LIN {X 0,Y 314.048,Z 563.182,A -85,B 0,C 180,E1 -16082.332,E2 -16082.332} C_VEL
LIN {X 0,Y 311.927,Z 573.073,A -85,B 0,C 180,E1 -16084.18,E2 -16084.18} C_VEL
LIN {X 0,Y 309.879,Z 582.152,A -85,B 0,C 180,E1 -16086.262,E2 -16086.262} C_VEL
LIN {X 0,Y 307.951,Z 590.287,A -85,B 0,C 180,E1 -16088.584,E2 -16088.584} C_VEL
LIN {X 0,Y 306.633,Z 595.997,A -85,B 0,C 180,E1 -16090.59,E2 -16090.59} C_VEL
LIN {X 0,Y 305.291,Z 601.948,A -85,B 0,C 180,E1 -16093.277,E2 -16093.277} C_VEL
LIN {X 0,Y 304.462,Z 606.083,A -85,B 0,C 180,E1 -16095.816,E2 -16095.816} C_VEL
LIN {X 0,Y 303.923,Z 608.604,A -85,B 0,C 180,E1 -16097.988,E2 -16097.988} C_VEL
LIN {X 0,Y 303.601,Z 610.421,A -85,B 0,C 180,E1 -16100.675,E2 -16100.675} C_VEL
LIN {X 0,Y 303.604,Z 610.898,A -85,B 0,C 180,E1 -16103.354,E2 -16103.354} C_VEL
LIN {X 0,Y 303.641,Z 610.642,A -85,B 0,C 180,E1 -16104.688,E2 -16104.688} C_VEL
LIN {X 0,Y 303.656,Z 609.146,A -85,B 0,C 180,E1 -16107.347,E2 -16107.347} C_VEL
LIN {X 0,Y 303.822,Z 606.306,A -85,B 0,C 180,E1 -16110,E2 -16110} C_VEL
LIN {X 0,Y 304.271,Z 602.046,A -85,B 0,C 180,E1 -16112.648,E2 -16112.648} C_VEL
LIN {X 0,Y 305.064,Z 596.235,A -85,B 0,C 180,E1 -16115.287,E2 -16115.287} C_VEL
LIN {X 0,Y 306.201,Z 589.686,A -85,B 0,C 180,E1 -16117.584,E2 -16117.584} C_VEL
LIN {X 0,Y 307.622,Z 581.561,A -85,B 0,C 180,E1 -16119.866,E2 -16119.866} C_VEL
LIN {X 0,Y 309.146,Z 572.018,A -85,B 0,C 180,E1 -16122.027,E2 -16122.027} C_VEL
LIN {X 0,Y 310.712,Z 562.821,A -85,B 0,C 180,E1 -16123.739,E2 -16123.739} C_VEL
LIN {X 0,Y 312.561,Z 551.345,A -85,B 0,C 180,E1 -16125.486,E2 -16125.486} C_VEL
LIN {X 0,Y 314.206,Z 539.898,A -85,B 0,C 180,E1 -16126.904,E2 -16126.904} C_VEL
LIN {X 0,Y 315.826,Z 527.334,A -85,B 0,C 180,E1 -16128.151,E2 -16128.151} C_VEL
LIN {X 0,Y 317.303,Z 514.341,A -85,B 0,C 180,E1 -16129.152,E2 -16129.152} C_VEL
LIN {X 0,Y 318.433,Z 500.352,A -85,B 0,C 180,E1 -16129.962,E2 -16129.962} C_VEL
LIN {X 0,Y 319.213,Z 486.734,A -85,B 0,C 180,E1 -16130.499,E2 -16130.499} C_VEL
LIN {X 0,Y 321.884,Z 387.028,A -85,B 0,C 180,E1 -16132.739,E2 -16132.739} C_VEL
LIN {X 0,Y 315.759,Z 371.085,A -85,B 0,C 180,E1 -16133.694,E2 -16133.694} C_VEL
LIN {X 0,Y 308.735,Z 355.109,A -85,B 0,C 180,E1 -16134.786,E2 -16134.786} C_VEL
LIN {X 0,Y 306.421,Z 349.762,A -85,B 0,C 180,E1 -16135.185,E2 -16135.185} C_VEL
LIN {X 0,Y 305.544,Z 346.052,A -85,B 0,C 180,E1 -16136.413,E2 -16136.413} C_VEL
LIN {X 0,Y 305.46,Z 346.061,A -85,B 0,C 180,E1 -16140.408,E2 -16140.408} C_VEL
LIN {X 0,Y 305.438,Z 346.062,A -85,B 0,C 180,E1 -16141.171,E2 -16141.171} C_VEL
LIN {X 0,Y 304.797,Z 346.144,A -85,B 0,C 180,E1 -16142.272,E2 -16142.272} C_VEL
LIN {X 0,Y 302.003,Z 346.49,A -85,B 0,C 180,E1 -16144.064,E2 -16144.064} C_VEL
LIN {X 0,Y 299.606,Z 346.785,A -85,B 0,C 180,E1 -16145.518,E2 -16145.518} C_VEL
LIN {X 0,Y 298.55,Z 346.917,A -85,B 0,C 180,E1 -16146.642,E2 -16146.642} C_VEL
LIN {X 0,Y 298.45,Z 346.93,A -85,B 0,C 180,E1 -16147.024,E2 -16147.024} C_VEL
LIN {X 0,Y 298.383,Z 346.926,A -85,B 0,C 180,E1 -16151.26,E2 -16151.26} C_VEL
LIN {X 0,Y 298.352,Z 346.941,A -85,B 0,C 180,E1 -16155.034,E2 -16155.034} C_VEL
LIN {X 0,Y 298.381,Z 346.935,A -85,B 0,C 180,E1 -16158.737,E2 -16158.737} C_VEL
LIN {X 0,Y 298.404,Z 346.93,A -85,B 0,C 180,E1 -16162.24,E2 -16162.24} C_VEL
LIN {X 0,Y 298.404,Z 346.935,A -85,B 0,C 180,E1 -16165.58,E2 -16165.58} C_VEL
LIN {X 0,Y 298.386,Z 346.941,A -85,B 0,C 180,E1 -16168.789,E2 -16168.789} C_VEL
LIN {X 0,Y 298.438,Z 346.919,A -85,B 0,C 180,E1 -16171.901,E2 -16171.901} C_VEL
LIN {X 0,Y 298.459,Z 346.929,A -85,B 0,C 180,E1 -16174.921,E2 -16174.921} C_VEL
LIN {X 0,Y 298.41,Z 346.918,A -85,B 0,C 180,E1 -16179.312,E2 -16179.312} C_VEL
LIN {X 0,Y 298.458,Z 346.927,A -85,B 0,C 180,E1 -16182.174,E2 -16182.174} C_VEL
LIN {X 0,Y 298.579,Z 346.911,A -85,B 0,C 180,E1 -16184.993,E2 -16184.993} C_VEL
LIN {X 0,Y 298.574,Z 346.907,A -85,B 0,C 180,E1 -16189.145,E2 -16189.145} C_VEL
LIN {X 0,Y 298.707,Z 346.9,A -85,B 0,C 180,E1 -16191.884,E2 -16191.884} C_VEL
LIN {X 0,Y 298.628,Z 346.89,A -85,B 0,C 180,E1 -16194.598,E2 -16194.598} C_VEL
LIN {X 0,Y 298.893,Z 346.877,A -85,B 0,C 180,E1 -16198.652,E2 -16198.652} C_VEL
LIN {X 0,Y 298.898,Z 346.872,A -85,B 0,C 180,E1 -16201.347,E2 -16201.347} C_VEL
LIN {X 0,Y 298.722,Z 346.899,A -85,B 0,C 180,E1 -16206.755,E2 -16206.755} C_VEL
LIN {X 0,Y 298.616,Z 346.897,A -85,B 0,C 180,E1 -16209.482,E2 -16209.482} C_VEL
LIN {X 0,Y 298.534,Z 346.922,A -85,B 0,C 180,E1 -16213.616,E2 -16213.616} C_VEL
LIN {X 0,Y 298.477,Z 346.92,A -85,B 0,C 180,E1 -16216.412,E2 -16216.412} C_VEL
LIN {X 0,Y 298.474,Z 346.929,A -85,B 0,C 180,E1 -16219.639,E2 -16219.639} C_VEL
LIN {X 0,Y 298.415,Z 346.935,A -85,B 0,C 180,E1 -16223.601,E2 -16223.601} C_VEL
LIN {X 0,Y 298.4,Z 346.931,A -85,B 0,C 180,E1 -16226.583,E2 -16226.583} C_VEL
LIN {X 0,Y 298.385,Z 346.937,A -85,B 0,C 180,E1 -16229.644,E2 -16229.644} C_VEL
LIN {X 0,Y 298.385,Z 346.94,A -85,B 0,C 180,E1 -16232.801,E2 -16232.801} C_VEL
LIN {X 0,Y 298.44,Z 346.932,A -85,B 0,C 180,E1 -16236.808,E2 -16236.808} C_VEL
LIN {X 0,Y 298.38,Z 346.928,A -85,B 0,C 180,E1 -16241.088,E2 -16241.088} C_VEL
LIN {X 0,Y 298.393,Z 346.937,A -85,B 0,C 180,E1 -16243.104,E2 -16243.104} C_VEL
LIN {X 0,Y 298.398,Z 346.939,A -85,B 0,C 180,E1 -16246.921,E2 -16246.921} C_VEL
LIN {X 0,Y 298.399,Z 346.946,A -85,B 0,C 180,E1 -16251.007,E2 -16251.007} C_VEL
LIN {X 0,Y 298.446,Z 347.048,A -85,B 0,C 180,E1 -16253.151,E2 -16253.151} C_VEL
LIN {X 0,Y 301.507,Z 359.563,A -85,B 0,C 180,E1 -16257.05,E2 -16257.05} C_VEL
LIN {X 0,Y 302.652,Z 364.595,A -85,B 0,C 180,E1 -16258.477,E2 -16258.477} C_VEL
LIN {X 0,Y 310.44,Z 383.686,A -85,B 0,C 180,E1 -16259.756,E2 -16259.756} C_VEL
LIN {X 0,Y 314.914,Z 411.594,A -85,B 0,C 180,E1 -16260.88,E2 -16260.88} C_VEL
LIN {X 0,Y 312.457,Z 500.646,A -85,B 0,C 180,E1 -16262.905,E2 -16262.905} C_VEL
LIN {X 0,Y 311.58,Z 514.525,A -85,B 0,C 180,E1 -16263.411,E2 -16263.411} C_VEL
LIN {X 0,Y 310.308,Z 528.189,A -85,B 0,C 180,E1 -16264.153,E2 -16264.153} C_VEL
LIN {X 0,Y 308.888,Z 541.031,A -85,B 0,C 180,E1 -16265.108,E2 -16265.108} C_VEL
LIN {X 0,Y 307.067,Z 554.478,A -85,B 0,C 180,E1 -16266.409,E2 -16266.409} C_VEL
LIN {X 0,Y 305.262,Z 566.32,A -85,B 0,C 180,E1 -16267.853,E2 -16267.853} C_VEL
LIN {X 0,Y 303.49,Z 576.274,A -85,B 0,C 180,E1 -16269.321,E2 -16269.321} C_VEL
LIN {X 0,Y 301.572,Z 587.25,A -85,B 0,C 180,E1 -16271.311,E2 -16271.311} C_VEL
LIN {X 0,Y 300.075,Z 596.312,A -85,B 0,C 180,E1 -16273.328,E2 -16273.328} C_VEL
LIN {X 0,Y 298.965,Z 603.853,A -85,B 0,C 180,E1 -16275.363,E2 -16275.363} C_VEL
LIN {X 0,Y 297.819,Z 611.042,A -85,B 0,C 180,E1 -16277.738,E2 -16277.738} C_VEL
LIN {X 0,Y 297.13,Z 616.051,A -85,B 0,C 180,E1 -16279.782,E2 -16279.782} C_VEL
LIN {X 0,Y 296.737,Z 621.214,A -85,B 0,C 180,E1 -16282.515,E2 -16282.515} C_VEL
LIN {X 0,Y 296.554,Z 624.106,A -85,B 0,C 180,E1 -16284.561,E2 -16284.561} C_VEL
LIN {X 0,Y 296.536,Z 626.656,A -85,B 0,C 180,E1 -16287.283,E2 -16287.283} C_VEL
LIN {X 0,Y 296.518,Z 627.833,A -85,B 0,C 180,E1 -16290,E2 -16290} C_VEL
LIN {X 0,Y 296.522,Z 627.671,A -85,B 0,C 180,E1 -16292.717,E2 -16292.717} C_VEL
LIN {X 0,Y 296.545,Z 626.116,A -85,B 0,C 180,E1 -16295.509,E2 -16295.509} C_VEL
LIN {X 0,Y 296.85,Z 623.32,A -85,B 0,C 180,E1 -16298.166,E2 -16298.166} C_VEL
LIN {X 0,Y 297.49,Z 619.034,A -85,B 0,C 180,E1 -16300.894,E2 -16300.894} C_VEL
LIN {X 0,Y 298.327,Z 614.817,A -85,B 0,C 180,E1 -16302.932,E2 -16302.932} C_VEL
LIN {X 0,Y 299.44,Z 609.647,A -85,B 0,C 180,E1 -16304.961,E2 -16304.961} C_VEL
LIN {X 0,Y 301.064,Z 602.238,A -85,B 0,C 180,E1 -16307.315,E2 -16307.315} C_VEL
LIN {X 0,Y 303.272,Z 593.049,A -85,B 0,C 180,E1 -16309.634,E2 -16309.634} C_VEL
LIN {X 0,Y 305.521,Z 583.471,A -85,B 0,C 180,E1 -16311.595,E2 -16311.595} C_VEL
LIN {X 0,Y 307.96,Z 572.871,A -85,B 0,C 180,E1 -16313.36,E2 -16313.36} C_VEL
LIN {X 0,Y 310.301,Z 561.536,A -85,B 0,C 180,E1 -16314.899,E2 -16314.899} C_VEL
LIN {X 0,Y 312.451,Z 549.755,A -85,B 0,C 180,E1 -16316.194,E2 -16316.194} C_VEL
LIN {X 0,Y 314.351,Z 537.392,A -85,B 0,C 180,E1 -16317.278,E2 -16317.278} C_VEL
LIN {X 0,Y 316.259,Z 523.679,A -85,B 0,C 180,E1 -16318.178,E2 -16318.178} C_VEL
LIN {X 0,Y 317.738,Z 509.393,A -85,B 0,C 180,E1 -16318.846,E2 -16318.846} C_VEL
LIN {X 0,Y 318.543,Z 494.481,A -85,B 0,C 180,E1 -16319.294,E2 -16319.294} C_VEL
LIN {X 0,Y 321.296,Z 414.11,A -85,B 0,C 180,E1 -16321.078,E2 -16321.078} C_VEL
LIN {X 0,Y 317.583,Z 394.103,A -85,B 0,C 180,E1 -16322.056,E2 -16322.056} C_VEL
LIN {X 0,Y 310.883,Z 379.558,A -85,B 0,C 180,E1 -16323.308,E2 -16323.308} C_VEL
LIN {X 0,Y 304.459,Z 366.874,A -85,B 0,C 180,E1 -16324.545,E2 -16324.545} C_VEL
LIN {X 0,Y 303.009,Z 363.713,A -85,B 0,C 180,E1 -16324.868,E2 -16324.868} C_VEL
LIN {X 0,Y 300.803,Z 355.353,A -85,B 0,C 180,E1 -16327.732,E2 -16327.732} C_VEL
LIN {X 0,Y 298.389,Z 346.922,A -85,B 0,C 180,E1 -16330.868,E2 -16330.868} C_VEL
LIN {X 0,Y 298.394,Z 346.931,A -85,B 0,C 180,E1 -16333.103,E2 -16333.103} C_VEL
LIN {X 0,Y 298.398,Z 346.935,A -85,B 0,C 180,E1 -16336.92,E2 -16336.92} C_VEL
LIN {X 0,Y 298.398,Z 346.941,A -85,B 0,C 180,E1 -16341.006,E2 -16341.006} C_VEL
LIN {X 0,Y 298.412,Z 346.941,A -85,B 0,C 180,E1 -16343.93,E2 -16343.93} C_VEL
LIN {X 0,Y 298.381,Z 346.932,A -85,B 0,C 180,E1 -16347.985,E2 -16347.985} C_VEL
LIN {X 0,Y 298.401,Z 346.924,A -85,B 0,C 180,E1 -16351.898,E2 -16351.898} C_VEL
LIN {X 0,Y 298.431,Z 346.929,A -85,B 0,C 180,E1 -16354.92,E2 -16354.92} C_VEL
LIN {X 0,Y 298.399,Z 346.94,A -85,B 0,C 180,E1 -16357.862,E2 -16357.862} C_VEL
LIN {X 0,Y 298.495,Z 346.926,A -85,B 0,C 180,E1 -16360.754,E2 -16360.754} C_VEL
LIN {X 0,Y 298.578,Z 346.913,A -85,B 0,C 180,E1 -16364.994,E2 -16364.994} C_VEL
LIN {X 0,Y 298.571,Z 346.91,A -85,B 0,C 180,E1 -16369.146,E2 -16369.146} C_VEL
LIN {X 0,Y 298.688,Z 346.898,A -85,B 0,C 180,E1 -16371.884,E2 -16371.884} C_VEL
LIN {X 0,Y 298.618,Z 346.91,A -85,B 0,C 180,E1 -16374.599,E2 -16374.599} C_VEL
LIN {X 0,Y 298.904,Z 346.869,A -85,B 0,C 180,E1 -16378.653,E2 -16378.653} C_VEL
LIN {X 0,Y 298.894,Z 346.874,A -85,B 0,C 180,E1 -16381.348,E2 -16381.348} C_VEL
LIN {X 0,Y 298.738,Z 346.89,A -85,B 0,C 180,E1 -16386.756,E2 -16386.756} C_VEL
LIN {X 0,Y 298.617,Z 346.915,A -85,B 0,C 180,E1 -16389.483,E2 -16389.483} C_VEL
LIN {X 0,Y 298.537,Z 346.923,A -85,B 0,C 180,E1 -16393.617,E2 -16393.617} C_VEL
LIN {X 0,Y 298.476,Z 346.921,A -85,B 0,C 180,E1 -16396.413,E2 -16396.413} C_VEL
LIN {X 0,Y 298.439,Z 346.931,A -85,B 0,C 180,E1 -16399.62,E2 -16399.62} C_VEL
LIN {X 0,Y 298.423,Z 346.933,A -85,B 0,C 180,E1 -16403.601,E2 -16403.601} C_VEL
LIN {X 0,Y 298.481,Z 346.932,A -85,B 0,C 180,E1 -16406.576,E2 -16406.576} C_VEL
LIN {X 0,Y 298.412,Z 346.938,A -85,B 0,C 180,E1 -16409.643,E2 -16409.643} C_VEL
LIN {X 0,Y 298.39,Z 346.942,A -85,B 0,C 180,E1 -16412.802,E2 -16412.802} C_VEL
LIN {X 0,Y 298.442,Z 346.929,A -85,B 0,C 180,E1 -16416.809,E2 -16416.809} C_VEL
LIN {X 0,Y 298.385,Z 346.943,A -85,B 0,C 180,E1 -16421.089,E2 -16421.089} C_VEL
LIN {X 0,Y 298.397,Z 346.939,A -85,B 0,C 180,E1 -16423.105,E2 -16423.105} C_VEL
LIN {X 0,Y 298.442,Z 347.061,A -85,B 0,C 180,E1 -16427.292,E2 -16427.292} C_VEL
LIN {X 0,Y 299.426,Z 350.748,A -85,B 0,C 180,E1 -16428.686,E2 -16428.686} C_VEL
LIN {X 0,Y 309.463,Z 368.66,A -85,B 0,C 180,E1 -16430.634,E2 -16430.634} C_VEL
LIN {X 0,Y 315.822,Z 381.45,A -85,B 0,C 180,E1 -16431.82,E2 -16431.82} C_VEL
LIN {X 0,Y 321.871,Z 395.005,A -85,B 0,C 180,E1 -16432.925,E2 -16432.925} C_VEL
LIN {X 0,Y 318.622,Z 487.207,A -85,B 0,C 180,E1 -16435.007,E2 -16435.007} C_VEL
LIN {X 0,Y 317.575,Z 501.841,A -85,B 0,C 180,E1 -16435.598,E2 -16435.598} C_VEL
LIN {X 0,Y 316.089,Z 515.831,A -85,B 0,C 180,E1 -16436.423,E2 -16436.423} C_VEL
LIN {X 0,Y 314.408,Z 527.939,A -85,B 0,C 180,E1 -16437.367,E2 -16437.367} C_VEL
LIN {X 0,Y 312.253,Z 540.703,A -85,B 0,C 180,E1 -16438.636,E2 -16438.636} C_VEL
LIN {X 0,Y 309.916,Z 552.287,A -85,B 0,C 180,E1 -16440.074,E2 -16440.074} C_VEL
LIN {X 0,Y 307.656,Z 562.893,A -85,B 0,C 180,E1 -16441.706,E2 -16441.706} C_VEL
LIN {X 0,Y 305.594,Z 572.086,A -85,B 0,C 180,E1 -16443.43,E2 -16443.43} C_VEL
LIN {X 0,Y 303.647,Z 580.667,A -85,B 0,C 180,E1 -16445.38,E2 -16445.38} C_VEL
LIN {X 0,Y 301.738,Z 588.045,A -85,B 0,C 180,E1 -16447.4,E2 -16447.4} C_VEL
LIN {X 0,Y 300.276,Z 594.164,A -85,B 0,C 180,E1 -16449.447,E2 -16449.447} C_VEL
LIN {X 0,Y 298.67,Z 600.637,A -85,B 0,C 180,E1 -16452.188,E2 -16452.188} C_VEL
LIN {X 0,Y 297.606,Z 605.444,A -85,B 0,C 180,E1 -16454.944,E2 -16454.944} C_VEL
LIN {X 0,Y 296.909,Z 608.73,A -85,B 0,C 180,E1 -16457.7,E2 -16457.7} C_VEL
LIN {X 0,Y 296.52,Z 610.594,A -85,B 0,C 180,E1 -16460.45,E2 -16460.45} C_VEL
LIN {X 0,Y 296.517,Z 611.111,A -85,B 0,C 180,E1 -16463.194,E2 -16463.194} C_VEL
LIN {X 0,Y 296.555,Z 610.874,A -85,B 0,C 180,E1 -16464.561,E2 -16464.561} C_VEL
LIN {X 0,Y 296.579,Z 609.417,A -85,B 0,C 180,E1 -16467.284,E2 -16467.284} C_VEL
LIN {X 0,Y 296.726,Z 606.619,A -85,B 0,C 180,E1 -16470,E2 -16470} C_VEL
LIN {X 0,Y 297.148,Z 603.624,A -85,B 0,C 180,E1 -16472.033,E2 -16472.033} C_VEL
LIN {X 0,Y 297.896,Z 598.23,A -85,B 0,C 180,E1 -16474.736,E2 -16474.736} C_VEL
LIN {X 0,Y 298.575,Z 593.122,A -85,B 0,C 180,E1 -16476.759,E2 -16476.759} C_VEL
LIN {X 0,Y 300.025,Z 585.752,A -85,B 0,C 180,E1 -16479.097,E2 -16479.097} C_VEL
LIN {X 0,Y 301.612,Z 576.798,A -85,B 0,C 180,E1 -16481.382,E2 -16481.382} C_VEL
LIN {X 0,Y 303.21,Z 567.089,A -85,B 0,C 180,E1 -16483.402,E2 -16483.402} C_VEL
LIN {X 0,Y 305.03,Z 556.516,A -85,B 0,C 180,E1 -16485.193,E2 -16485.193} C_VEL
LIN {X 0,Y 306.934,Z 544.818,A -85,B 0,C 180,E1 -16486.802,E2 -16486.802} C_VEL
LIN {X 0,Y 308.525,Z 533.376,A -85,B 0,C 180,E1 -16488.081,E2 -16488.081} C_VEL
LIN {X 0,Y 310.089,Z 520.948,A -85,B 0,C 180,E1 -16489.185,E2 -16489.185} C_VEL
LIN {X 0,Y 311.431,Z 507.132,A -85,B 0,C 180,E1 -16490.129,E2 -16490.129} C_VEL
LIN {X 0,Y 312.498,Z 493.489,A -85,B 0,C 180,E1 -16490.788,E2 -16490.788} C_VEL
LIN {X 0,Y 313.003,Z 479.899,A -85,B 0,C 180,E1 -16491.222,E2 -16491.222} C_VEL
LIN {X 0,Y 315.427,Z 388.282,A -85,B 0,C 180,E1 -16493.293,E2 -16493.293} C_VEL
LIN {X 0,Y 307.234,Z 367.72,A -85,B 0,C 180,E1 -16494.609,E2 -16494.609} C_VEL
LIN {X 0,Y 299.236,Z 349.982,A -85,B 0,C 180,E1 -16495.937,E2 -16495.937} C_VEL
LIN {X 0,Y 298.479,Z 346.931,A -85,B 0,C 180,E1 -16497.018,E2 -16497.018} C_VEL
LIN {X 0,Y 298.393,Z 346.94,A -85,B 0,C 180,E1 -16501.208,E2 -16501.208} C_VEL
LIN {X 0,Y 298.428,Z 346.933,A -85,B 0,C 180,E1 -16504.486,E2 -16504.486} C_VEL
LIN {X 0,Y 298.45,Z 346.93,A -85,B 0,C 180,E1 -16507.024,E2 -16507.024} C_VEL
LIN {X 0,Y 297.738,Z 347.023,A -85,B 0,C 180,E1 -16508.15,E2 -16508.15} C_VEL
LIN {X 0,Y 294.851,Z 347.382,A -85,B 0,C 180,E1 -16509.983,E2 -16509.983} C_VEL
LIN {X 0,Y 292.426,Z 347.682,A -85,B 0,C 180,E1 -16511.47,E2 -16511.47} C_VEL
LIN {X 0,Y 291.385,Z 347.812,A -85,B 0,C 180,E1 -16512.623,E2 -16512.623} C_VEL
LIN {X 0,Y 291.299,Z 347.821,A -85,B 0,C 180,E1 -16513.013,E2 -16513.013} C_VEL
LIN {X 0,Y 291.317,Z 347.818,A -85,B 0,C 180,E1 -16517.506,E2 -16517.506} C_VEL
LIN {X 0,Y 291.344,Z 347.817,A -85,B 0,C 180,E1 -16521.156,E2 -16521.156} C_VEL
LIN {X 0,Y 291.357,Z 347.817,A -85,B 0,C 180,E1 -16524.625,E2 -16524.625} C_VEL
LIN {X 0,Y 291.366,Z 347.814,A -85,B 0,C 180,E1 -16527.949,E2 -16527.949} C_VEL
LIN {X 0,Y 291.365,Z 347.805,A -85,B 0,C 180,E1 -16531.156,E2 -16531.156} C_VEL
LIN {X 0,Y 291.394,Z 347.805,A -85,B 0,C 180,E1 -16534.269,E2 -16534.269} C_VEL
LIN {X 0,Y 291.361,Z 347.811,A -85,B 0,C 180,E1 -16537.297,E2 -16537.297} C_VEL
LIN {X 0,Y 291.384,Z 347.793,A -85,B 0,C 180,E1 -16540.264,E2 -16540.264} C_VEL
LIN {X 0,Y 291.491,Z 347.797,A -85,B 0,C 180,E1 -16544.664,E2 -16544.664} C_VEL
LIN {X 0,Y 291.52,Z 347.782,A -85,B 0,C 180,E1 -16548.879,E2 -16548.879} C_VEL
LIN {X 0,Y 291.658,Z 347.778,A -85,B 0,C 180,E1 -16551.687,E2 -16551.687} C_VEL
LIN {X 0,Y 291.598,Z 347.766,A -85,B 0,C 180,E1 -16554.467,E2 -16554.467} C_VEL
LIN {X 0,Y 291.861,Z 347.752,A -85,B 0,C 180,E1 -16558.62,E2 -16558.62} C_VEL
LIN {X 0,Y 291.864,Z 347.748,A -85,B 0,C 180,E1 -16561.379,E2 -16561.379} C_VEL
LIN {X 0,Y 291.675,Z 347.776,A -85,B 0,C 180,E1 -16566.919,E2 -16566.919} C_VEL
LIN {X 0,Y 291.559,Z 347.776,A -85,B 0,C 180,E1 -16569.714,E2 -16569.714} C_VEL
LIN {X 0,Y 291.505,Z 347.796,A -85,B 0,C 180,E1 -16573.951,E2 -16573.951} C_VEL
LIN {X 0,Y 291.431,Z 347.802,A -85,B 0,C 180,E1 -16576.821,E2 -16576.821} C_VEL
LIN {X 0,Y 291.416,Z 347.804,A -85,B 0,C 180,E1 -16579.86,E2 -16579.86} C_VEL
LIN {X 0,Y 291.355,Z 347.815,A -85,B 0,C 180,E1 -16584.209,E2 -16584.209} C_VEL
LIN {X 0,Y 291.346,Z 347.813,A -85,B 0,C 180,E1 -16587.279,E2 -16587.279} C_VEL
LIN {X 0,Y 291.31,Z 347.815,A -85,B 0,C 180,E1 -16590.44,E2 -16590.44} C_VEL
LIN {X 0,Y 291.336,Z 347.816,A -85,B 0,C 180,E1 -16593.699,E2 -16593.699} C_VEL
LIN {X 0,Y 291.369,Z 347.812,A -85,B 0,C 180,E1 -16597.254,E2 -16597.254} C_VEL
LIN {X 0,Y 291.326,Z 347.809,A -85,B 0,C 180,E1 -16600.643,E2 -16600.643} C_VEL
LIN {X 0,Y 291.285,Z 347.825,A -85,B 0,C 180,E1 -16604.403,E2 -16604.403} C_VEL
LIN {X 0,Y 291.321,Z 347.822,A -85,B 0,C 180,E1 -16608.405,E2 -16608.405} C_VEL
LIN {X 0,Y 291.359,Z 347.823,A -85,B 0,C 180,E1 -16612.017,E2 -16612.017} C_VEL
LIN {X 0,Y 291.394,Z 348.003,A -85,B 0,C 180,E1 -16612.552,E2 -16612.552} C_VEL
LIN {X 0,Y 293.885,Z 358.064,A -85,B 0,C 180,E1 -16615.809,E2 -16615.809} C_VEL
LIN {X 0,Y 295.347,Z 364.294,A -85,B 0,C 180,E1 -16617.686,E2 -16617.686} C_VEL
LIN {X 0,Y 303.462,Z 383.711,A -85,B 0,C 180,E1 -16619.066,E2 -16619.066} C_VEL
LIN {X 0,Y 304.714,Z 387.787,A -85,B 0,C 180,E1 -16619.3,E2 -16619.3} C_VEL
LIN {X 0,Y 308.592,Z 413.856,A -85,B 0,C 180,E1 -16620.352,E2 -16620.352} C_VEL
LIN {X 0,Y 305.941,Z 502.681,A -85,B 0,C 180,E1 -16622.418,E2 -16622.418} C_VEL
LIN {X 0,Y 304.99,Z 516.506,A -85,B 0,C 180,E1 -16622.975,E2 -16622.975} C_VEL
LIN {X 0,Y 303.509,Z 530.662,A -85,B 0,C 180,E1 -16623.807,E2 -16623.807} C_VEL
LIN {X 0,Y 301.908,Z 543.792,A -85,B 0,C 180,E1 -16624.861,E2 -16624.861} C_VEL
LIN {X 0,Y 300.102,Z 556.583,A -85,B 0,C 180,E1 -16626.184,E2 -16626.184} C_VEL
LIN {X 0,Y 298.23,Z 568.081,A -85,B 0,C 180,E1 -16627.667,E2 -16627.667} C_VEL
LIN {X 0,Y 296.42,Z 577.703,A -85,B 0,C 180,E1 -16629.168,E2 -16629.168} C_VEL
LIN {X 0,Y 294.49,Z 588.41,A -85,B 0,C 180,E1 -16631.206,E2 -16631.206} C_VEL
LIN {X 0,Y 292.967,Z 597.244,A -85,B 0,C 180,E1 -16633.27,E2 -16633.27} C_VEL
LIN {X 0,Y 291.827,Z 604.586,A -85,B 0,C 180,E1 -16635.353,E2 -16635.353} C_VEL
LIN {X 0,Y 290.848,Z 610.685,A -85,B 0,C 180,E1 -16637.44,E2 -16637.44} C_VEL
LIN {X 0,Y 290.091,Z 615.727,A -85,B 0,C 180,E1 -16639.531,E2 -16639.531} C_VEL
LIN {X 0,Y 289.669,Z 620.922,A -85,B 0,C 180,E1 -16642.332,E2 -16642.332} C_VEL
LIN {X 0,Y 289.477,Z 623.927,A -85,B 0,C 180,E1 -16644.505,E2 -16644.505} C_VEL
LIN {X 0,Y 289.44,Z 626.42,A -85,B 0,C 180,E1 -16647.217,E2 -16647.217} C_VEL
LIN {X 0,Y 289.436,Z 627.625,A -85,B 0,C 180,E1 -16650,E2 -16650} C_VEL
LIN {X 0,Y 289.426,Z 627.489,A -85,B 0,C 180,E1 -16652.784,E2 -16652.784} C_VEL
LIN {X 0,Y 289.475,Z 626.019,A -85,B 0,C 180,E1 -16655.573,E2 -16655.573} C_VEL
LIN {X 0,Y 289.779,Z 623.193,A -85,B 0,C 180,E1 -16658.367,E2 -16658.367} C_VEL
LIN {X 0,Y 290.457,Z 618.937,A -85,B 0,C 180,E1 -16661.161,E2 -16661.161} C_VEL
LIN {X 0,Y 291.781,Z 613.133,A -85,B 0,C 180,E1 -16663.937,E2 -16663.937} C_VEL
LIN {X 0,Y 293.346,Z 605.905,A -85,B 0,C 180,E1 -16666.601,E2 -16666.601} C_VEL
LIN {X 0,Y 295.174,Z 598.554,A -85,B 0,C 180,E1 -16668.749,E2 -16668.749} C_VEL
LIN {X 0,Y 297.284,Z 590.133,A -85,B 0,C 180,E1 -16670.769,E2 -16670.769} C_VEL
LIN {X 0,Y 299.826,Z 580.006,A -85,B 0,C 180,E1 -16672.753,E2 -16672.753} C_VEL
LIN {X 0,Y 302.443,Z 568.683,A -85,B 0,C 180,E1 -16674.542,E2 -16674.542} C_VEL
LIN {X 0,Y 304.735,Z 557.452,A -85,B 0,C 180,E1 -16675.988,E2 -16675.988} C_VEL
LIN {X 0,Y 306.912,Z 545.21,A -85,B 0,C 180,E1 -16677.256,E2 -16677.256} C_VEL
LIN {X 0,Y 309.078,Z 531.593,A -85,B 0,C 180,E1 -16678.337,E2 -16678.337} C_VEL
LIN {X 0,Y 310.924,Z 517.265,A -85,B 0,C 180,E1 -16679.168,E2 -16679.168} C_VEL
LIN {X 0,Y 312.168,Z 503.064,A -85,B 0,C 180,E1 -16679.733,E2 -16679.733} C_VEL
LIN {X 0,Y 313.436,Z 469.222,A -85,B 0,C 180,E1 -16680.542,E2 -16680.542} C_VEL
LIN {X 0,Y 315.373,Z 415.215,A -85,B 0,C 180,E1 -16681.759,E2 -16681.759} C_VEL
LIN {X 0,Y 312.107,Z 397.239,A -85,B 0,C 180,E1 -16682.659,E2 -16682.659} C_VEL
LIN {X 0,Y 304.554,Z 380.759,A -85,B 0,C 180,E1 -16684.131,E2 -16684.131} C_VEL
LIN {X 0,Y 297.376,Z 366.86,A -85,B 0,C 180,E1 -16685.576,E2 -16685.576} C_VEL
LIN {X 0,Y 295.743,Z 363.497,A -85,B 0,C 180,E1 -16685.942,E2 -16685.942} C_VEL
LIN {X 0,Y 293.152,Z 354.119,A -85,B 0,C 180,E1 -16689.326,E2 -16689.326} C_VEL
LIN {X 0,Y 291.327,Z 347.81,A -85,B 0,C 180,E1 -16691.794,E2 -16691.794} C_VEL
LIN {X 0,Y 291.285,Z 347.818,A -85,B 0,C 180,E1 -16695.597,E2 -16695.597} C_VEL
LIN {X 0,Y 291.327,Z 347.818,A -85,B 0,C 180,E1 -16699.357,E2 -16699.357} C_VEL
LIN {X 0,Y 291.401,Z 347.809,A -85,B 0,C 180,E1 -16702.919,E2 -16702.919} C_VEL
LIN {X 0,Y 291.337,Z 347.819,A -85,B 0,C 180,E1 -16706.301,E2 -16706.301} C_VEL
LIN {X 0,Y 291.331,Z 347.787,A -85,B 0,C 180,E1 -16710.277,E2 -16710.277} C_VEL
LIN {X 0,Y 291.351,Z 347.814,A -85,B 0,C 180,E1 -16714.266,E2 -16714.266} C_VEL
LIN {X 0,Y 291.359,Z 347.816,A -85,B 0,C 180,E1 -16717.298,E2 -16717.298} C_VEL
LIN {X 0,Y 291.432,Z 347.802,A -85,B 0,C 180,E1 -16720.269,E2 -16720.269} C_VEL
LIN {X 0,Y 291.49,Z 347.795,A -85,B 0,C 180,E1 -16724.665,E2 -16724.665} C_VEL
LIN {X 0,Y 291.517,Z 347.787,A -85,B 0,C 180,E1 -16728.88,E2 -16728.88} C_VEL
LIN {X 0,Y 291.642,Z 347.777,A -85,B 0,C 180,E1 -16731.687,E2 -16731.687} C_VEL
LIN {X 0,Y 291.588,Z 347.786,A -85,B 0,C 180,E1 -16734.468,E2 -16734.468} C_VEL
LIN {X 0,Y 291.87,Z 347.745,A -85,B 0,C 180,E1 -16738.621,E2 -16738.621} C_VEL
LIN {X 0,Y 291.862,Z 347.749,A -85,B 0,C 180,E1 -16741.38,E2 -16741.38} C_VEL
LIN {X 0,Y 291.69,Z 347.767,A -85,B 0,C 180,E1 -16746.92,E2 -16746.92} C_VEL
LIN {X 0,Y 291.56,Z 347.792,A -85,B 0,C 180,E1 -16749.715,E2 -16749.715} C_VEL
LIN {X 0,Y 291.507,Z 347.798,A -85,B 0,C 180,E1 -16753.952,E2 -16753.952} C_VEL
LIN {X 0,Y 291.421,Z 347.8,A -85,B 0,C 180,E1 -16756.822,E2 -16756.822} C_VEL
LIN {X 0,Y 291.385,Z 347.809,A -85,B 0,C 180,E1 -16759.843,E2 -16759.843} C_VEL
LIN {X 0,Y 291.377,Z 347.808,A -85,B 0,C 180,E1 -16764.208,E2 -16764.208} C_VEL
LIN {X 0,Y 291.415,Z 347.806,A -85,B 0,C 180,E1 -16767.273,E2 -16767.273} C_VEL
LIN {X 0,Y 291.329,Z 347.819,A -85,B 0,C 180,E1 -16770.438,E2 -16770.438} C_VEL
LIN {X 0,Y 291.34,Z 347.817,A -85,B 0,C 180,E1 -16773.7,E2 -16773.7} C_VEL
LIN {X 0,Y 291.372,Z 347.808,A -85,B 0,C 180,E1 -16777.255,E2 -16777.255} C_VEL
LIN {X 0,Y 291.33,Z 347.817,A -85,B 0,C 180,E1 -16780.644,E2 -16780.644} C_VEL
LIN {X 0,Y 291.288,Z 347.824,A -85,B 0,C 180,E1 -16784.403,E2 -16784.403} C_VEL
LIN {X 0,Y 291.332,Z 347.933,A -85,B 0,C 180,E1 -16786.363,E2 -16786.363} C_VEL
LIN {X 0,Y 292.176,Z 350.843,A -85,B 0,C 180,E1 -16787.563,E2 -16787.563} C_VEL
LIN {X 0,Y 294.625,Z 355.1,A -85,B 0,C 180,E1 -16788.083,E2 -16788.083} C_VEL
LIN {X 0,Y 303.961,Z 371.708,A -85,B 0,C 180,E1 -16789.962,E2 -16789.962} C_VEL
LIN {X 0,Y 311.045,Z 386.056,A -85,B 0,C 180,E1 -16791.332,E2 -16791.332} C_VEL
LIN {X 0,Y 315.946,Z 397.109,A -85,B 0,C 180,E1 -16792.26,E2 -16792.26} C_VEL
LIN {X 0,Y 312.609,Z 487.449,A -85,B 0,C 180,E1 -16794.331,E2 -16794.331} C_VEL
LIN {X 0,Y 311.512,Z 502.065,A -85,B 0,C 180,E1 -16794.93,E2 -16794.93} C_VEL
LIN {X 0,Y 309.958,Z 516.045,A -85,B 0,C 180,E1 -16795.765,E2 -16795.765} C_VEL
LIN {X 0,Y 308.072,Z 529.041,A -85,B 0,C 180,E1 -16796.805,E2 -16796.805} C_VEL
LIN {X 0,Y 305.86,Z 541.63,A -85,B 0,C 180,E1 -16798.097,E2 -16798.097} C_VEL
LIN {X 0,Y 303.424,Z 553.083,A -85,B 0,C 180,E1 -16799.558,E2 -16799.558} C_VEL
LIN {X 0,Y 301.307,Z 562.604,A -85,B 0,C 180,E1 -16801.054,E2 -16801.054} C_VEL
LIN {X 0,Y 298.815,Z 573.192,A -85,B 0,C 180,E1 -16803.08,E2 -16803.08} C_VEL
LIN {X 0,Y 296.73,Z 581.893,A -85,B 0,C 180,E1 -16805.141,E2 -16805.141} C_VEL
LIN {X 0,Y 294.506,Z 590.186,A -85,B 0,C 180,E1 -16807.554,E2 -16807.554} C_VEL
LIN {X 0,Y 292.943,Z 596.187,A -85,B 0,C 180,E1 -16809.736,E2 -16809.736} C_VEL
LIN {X 0,Y 291.455,Z 602.043,A -85,B 0,C 180,E1 -16812.458,E2 -16812.458} C_VEL
LIN {X 0,Y 290.647,Z 605.514,A -85,B 0,C 180,E1 -16814.575,E2 -16814.575} C_VEL
LIN {X 0,Y 289.873,Z 608.849,A -85,B 0,C 180,E1 -16817.397,E2 -16817.397} C_VEL
LIN {X 0,Y 289.453,Z 610.765,A -85,B 0,C 180,E1 -16820.215,E2 -16820.215} C_VEL
LIN {X 0,Y 289.425,Z 611.324,A -85,B 0,C 180,E1 -16823.027,E2 -16823.027} C_VEL
LIN {X 0,Y 289.484,Z 611.08,A -85,B 0,C 180,E1 -16824.502,E2 -16824.502} C_VEL
LIN {X 0,Y 289.504,Z 609.688,A -85,B 0,C 180,E1 -16827.217,E2 -16827.217} C_VEL
LIN {X 0,Y 289.632,Z 606.932,A -85,B 0,C 180,E1 -16830,E2 -16830} C_VEL
LIN {X 0,Y 290.056,Z 603.967,A -85,B 0,C 180,E1 -16832.083,E2 -16832.083} C_VEL
LIN {X 0,Y 290.838,Z 598.631,A -85,B 0,C 180,E1 -16834.852,E2 -16834.852} C_VEL
LIN {X 0,Y 291.544,Z 593.547,A -85,B 0,C 180,E1 -16836.923,E2 -16836.923} C_VEL
LIN {X 0,Y 293.052,Z 586.243,A -85,B 0,C 180,E1 -16839.316,E2 -16839.316} C_VEL
LIN {X 0,Y 294.671,Z 577.506,A -85,B 0,C 180,E1 -16841.62,E2 -16841.62} C_VEL
LIN {X 0,Y 296.338,Z 567.729,A -85,B 0,C 180,E1 -16843.719,E2 -16843.719} C_VEL
LIN {X 0,Y 298.231,Z 557.244,A -85,B 0,C 180,E1 -16845.548,E2 -16845.548} C_VEL
LIN {X 0,Y 300.205,Z 545.653,A -85,B 0,C 180,E1 -16847.191,E2 -16847.191} C_VEL
LIN {X 0,Y 301.83,Z 534.356,A -85,B 0,C 180,E1 -16848.496,E2 -16848.496} C_VEL
LIN {X 0,Y 303.444,Z 522.127,A -85,B 0,C 180,E1 -16849.622,E2 -16849.622} C_VEL
LIN {X 0,Y 304.854,Z 508.609,A -85,B 0,C 180,E1 -16850.583,E2 -16850.583} C_VEL
LIN {X 0,Y 305.993,Z 494.584,A -85,B 0,C 180,E1 -16851.295,E2 -16851.295} C_VEL
LIN {X 0,Y 306.59,Z 479.926,A -85,B 0,C 180,E1 -16851.781,E2 -16851.781} C_VEL
LIN {X 0,Y 309.064,Z 389.998,A -85,B 0,C 180,E1 -16853.852,E2 -16853.852} C_VEL
LIN {X 0,Y 301.47,Z 370.915,A -85,B 0,C 180,E1 -16855.115,E2 -16855.115} C_VEL
LIN {X 0,Y 293.551,Z 353.546,A -85,B 0,C 180,E1 -16856.448,E2 -16856.448} C_VEL
LIN {X 0,Y 291.983,Z 350.18,A -85,B 0,C 180,E1 -16856.749,E2 -16856.749} C_VEL
LIN {X 0,Y 291.45,Z 347.807,A -85,B 0,C 180,E1 -16857.657,E2 -16857.657} C_VEL
LIN {X 0,Y 291.372,Z 347.816,A -85,B 0,C 180,E1 -16862.048,E2 -16862.048} C_VEL
LIN {X 0,Y 291.385,Z 347.803,A -85,B 0,C 180,E1 -16865.369,E2 -16865.369} C_VEL
LIN {X 0,Y 291.364,Z 347.81,A -85,B 0,C 180,E1 -16868.838,E2 -16868.838} C_VEL
LIN {X 0,Y 291.299,Z 347.821,A -85,B 0,C 180,E1 -16873.013,E2 -16873.013} C_VEL
LIN {X 0,Y 290.623,Z 347.908,A -85,B 0,C 180,E1 -16874.166,E2 -16874.166} C_VEL
LIN {X 0,Y 287.754,Z 348.266,A -85,B 0,C 180,E1 -16876.044,E2 -16876.044} C_VEL
LIN {X 0,Y 285.338,Z 348.562,A -85,B 0,C 180,E1 -16877.568,E2 -16877.568} C_VEL
LIN {X 0,Y 284.322,Z 348.686,A -85,B 0,C 180,E1 -16878.75,E2 -16878.75} C_VEL
LIN {X 0,Y 284.249,Z 348.694,A -85,B 0,C 180,E1 -16879.15,E2 -16879.15} C_VEL
LIN {X 0,Y 284.315,Z 348.685,A -85,B 0,C 180,E1 -16882.278,E2 -16882.278} C_VEL
LIN {X 0,Y 284.304,Z 348.693,A -85,B 0,C 180,E1 -16885.349,E2 -16885.349} C_VEL
LIN {X 0,Y 284.289,Z 348.697,A -85,B 0,C 180,E1 -16888.724,E2 -16888.724} C_VEL
LIN {X 0,Y 284.31,Z 348.678,A -85,B 0,C 180,E1 -16891.986,E2 -16891.986} C_VEL
LIN {X 0,Y 284.322,Z 348.692,A -85,B 0,C 180,E1 -16895.151,E2 -16895.151} C_VEL
LIN {X 0,Y 284.302,Z 348.685,A -85,B 0,C 180,E1 -16898.234,E2 -16898.234} C_VEL
LIN {X 0,Y 284.325,Z 348.681,A -85,B 0,C 180,E1 -16901.256,E2 -16901.256} C_VEL
LIN {X 0,Y 284.455,Z 348.666,A -85,B 0,C 180,E1 -16905.695,E2 -16905.695} C_VEL
LIN {X 0,Y 284.506,Z 348.665,A -85,B 0,C 180,E1 -16910.042,E2 -16910.042} C_VEL
LIN {X 0,Y 284.649,Z 348.646,A -85,B 0,C 180,E1 -16912.908,E2 -16912.908} C_VEL
LIN {X 0,Y 284.829,Z 348.628,A -85,B 0,C 180,E1 -16918.586,E2 -16918.586} C_VEL
LIN {X 0,Y 284.83,Z 348.624,A -85,B 0,C 180,E1 -16921.413,E2 -16921.413} C_VEL
LIN {X 0,Y 284.631,Z 348.653,A -85,B 0,C 180,E1 -16927.091,E2 -16927.091} C_VEL
LIN {X 0,Y 284.505,Z 348.655,A -85,B 0,C 180,E1 -16929.957,E2 -16929.957} C_VEL
LIN {X 0,Y 284.454,Z 348.67,A -85,B 0,C 180,E1 -16934.304,E2 -16934.304} C_VEL
LIN {X 0,Y 284.365,Z 348.686,A -85,B 0,C 180,E1 -16938.741,E2 -16938.741} C_VEL
LIN {X 0,Y 284.303,Z 348.682,A -85,B 0,C 180,E1 -16941.765,E2 -16941.765} C_VEL
LIN {X 0,Y 284.3,Z 348.69,A -85,B 0,C 180,E1 -16944.85,E2 -16944.85} C_VEL
LIN {X 0,Y 284.276,Z 348.698,A -85,B 0,C 180,E1 -16948.016,E2 -16948.016} C_VEL
LIN {X 0,Y 284.277,Z 348.694,A -85,B 0,C 180,E1 -16951.276,E2 -16951.276} C_VEL
LIN {X 0,Y 284.335,Z 348.69,A -85,B 0,C 180,E1 -16955.348,E2 -16955.348} C_VEL
LIN {X 0,Y 284.306,Z 348.695,A -85,B 0,C 180,E1 -16958.17,E2 -16958.17} C_VEL
LIN {X 0,Y 284.263,Z 348.687,A -85,B 0,C 180,E1 -16962.125,E2 -16962.125} C_VEL
LIN {X 0,Y 284.251,Z 348.703,A -85,B 0,C 180,E1 -16966.19,E2 -16966.19} C_VEL
LIN {X 0,Y 284.302,Z 348.699,A -85,B 0,C 180,E1 -16970.025,E2 -16970.025} C_VEL
LIN {X 0,Y 284.323,Z 348.799,A -85,B 0,C 180,E1 -16971.869,E2 -16971.869} C_VEL
LIN {X 0,Y 286.905,Z 359.031,A -85,B 0,C 180,E1 -16975.298,E2 -16975.298} C_VEL
LIN {X 0,Y 288.07,Z 363.925,A -85,B 0,C 180,E1 -16976.85,E2 -16976.85} C_VEL
LIN {X 0,Y 297.123,Z 385.291,A -85,B 0,C 180,E1 -16978.45,E2 -16978.45} C_VEL
LIN {X 0,Y 298.619,Z 389.86,A -85,B 0,C 180,E1 -16978.731,E2 -16978.731} C_VEL
LIN {X 0,Y 302.237,Z 413.709,A -85,B 0,C 180,E1 -16979.733,E2 -16979.733} C_VEL
LIN {X 0,Y 299.564,Z 502.046,A -85,B 0,C 180,E1 -16981.827,E2 -16981.827} C_VEL
LIN {X 0,Y 298.547,Z 516.014,A -85,B 0,C 180,E1 -16982.39,E2 -16982.39} C_VEL
LIN {X 0,Y 297.134,Z 529.683,A -85,B 0,C 180,E1 -16983.201,E2 -16983.201} C_VEL
LIN {X 0,Y 295.469,Z 542.982,A -85,B 0,C 180,E1 -16984.273,E2 -16984.273} C_VEL
LIN {X 0,Y 293.616,Z 555.545,A -85,B 0,C 180,E1 -16985.579,E2 -16985.579} C_VEL
LIN {X 0,Y 291.841,Z 566.288,A -85,B 0,C 180,E1 -16986.964,E2 -16986.964} C_VEL
LIN {X 0,Y 289.717,Z 577.161,A -85,B 0,C 180,E1 -16988.662,E2 -16988.662} C_VEL
LIN {X 0,Y 287.711,Z 587.925,A -85,B 0,C 180,E1 -16990.746,E2 -16990.746} C_VEL
LIN {X 0,Y 286.116,Z 596.807,A -85,B 0,C 180,E1 -16992.857,E2 -16992.857} C_VEL
LIN {X 0,Y 284.687,Z 605.317,A -85,B 0,C 180,E1 -16995.343,E2 -16995.343} C_VEL
LIN {X 0,Y 283.548,Z 612.153,A -85,B 0,C 180,E1 -16997.838,E2 -16997.838} C_VEL
LIN {X 0,Y 282.902,Z 616.843,A -85,B 0,C 180,E1 -16999.986,E2 -16999.986} C_VEL
LIN {X 0,Y 282.502,Z 621.703,A -85,B 0,C 180,E1 -17002.855,E2 -17002.855} C_VEL
LIN {X 0,Y 282.336,Z 625.047,A -85,B 0,C 180,E1 -17005.717,E2 -17005.717} C_VEL
LIN {X 0,Y 282.34,Z 626.969,A -85,B 0,C 180,E1 -17008.574,E2 -17008.574} C_VEL
LIN {X 0,Y 282.334,Z 627.529,A -85,B 0,C 180,E1 -17011.426,E2 -17011.426} C_VEL
LIN {X 0,Y 282.299,Z 626.752,A -85,B 0,C 180,E1 -17014.283,E2 -17014.283} C_VEL
LIN {X 0,Y 282.495,Z 624.638,A -85,B 0,C 180,E1 -17017.145,E2 -17017.145} C_VEL
LIN {X 0,Y 283.053,Z 621.139,A -85,B 0,C 180,E1 -17020.009,E2 -17020.009} C_VEL
LIN {X 0,Y 284.043,Z 616.156,A -85,B 0,C 180,E1 -17022.866,E2 -17022.866} C_VEL
LIN {X 0,Y 285.235,Z 611.366,A -85,B 0,C 180,E1 -17024.993,E2 -17024.993} C_VEL
LIN {X 0,Y 286.878,Z 604.459,A -85,B 0,C 180,E1 -17027.463,E2 -17027.463} C_VEL
LIN {X 0,Y 289.155,Z 595.915,A -85,B 0,C 180,E1 -17029.893,E2 -17029.893} C_VEL
LIN {X 0,Y 291.48,Z 587.015,A -85,B 0,C 180,E1 -17031.945,E2 -17031.945} C_VEL
LIN {X 0,Y 294.236,Z 576.256,A -85,B 0,C 180,E1 -17033.957,E2 -17033.957} C_VEL
LIN {X 0,Y 296.841,Z 565.211,A -85,B 0,C 180,E1 -17035.626,E2 -17035.626} C_VEL
LIN {X 0,Y 299.25,Z 553.486,A -85,B 0,C 180,E1 -17037.066,E2 -17037.066} C_VEL
LIN {X 0,Y 301.285,Z 542.106,A -85,B 0,C 180,E1 -17038.187,E2 -17038.187} C_VEL
LIN {X 0,Y 303.39,Z 528.806,A -85,B 0,C 180,E1 -17039.202,E2 -17039.202} C_VEL
LIN {X 0,Y 305.118,Z 515.093,A -85,B 0,C 180,E1 -17039.969,E2 -17039.969} C_VEL
LIN {X 0,Y 306.294,Z 500.988,A -85,B 0,C 180,E1 -17040.504,E2 -17040.504} C_VEL
LIN {X 0,Y 309.442,Z 416.086,A -85,B 0,C 180,E1 -17042.481,E2 -17042.481} C_VEL
LIN {X 0,Y 306.483,Z 399.885,A -85,B 0,C 180,E1 -17043.322,E2 -17043.322} C_VEL
LIN {X 0,Y 299.485,Z 384.622,A -85,B 0,C 180,E1 -17044.737,E2 -17044.737} C_VEL
LIN {X 0,Y 292.373,Z 370.74,A -85,B 0,C 180,E1 -17046.225,E2 -17046.225} C_VEL
LIN {X 0,Y 288.443,Z 363.215,A -85,B 0,C 180,E1 -17047.109,E2 -17047.109} C_VEL
LIN {X 0,Y 285.713,Z 353.446,A -85,B 0,C 180,E1 -17050.819,E2 -17050.819} C_VEL
LIN {X 0,Y 284.257,Z 348.692,A -85,B 0,C 180,E1 -17052.802,E2 -17052.802} C_VEL
LIN {X 0,Y 284.251,Z 348.699,A -85,B 0,C 180,E1 -17056.189,E2 -17056.189} C_VEL
LIN {X 0,Y 284.301,Z 348.692,A -85,B 0,C 180,E1 -17060.023,E2 -17060.023} C_VEL
LIN {X 0,Y 284.326,Z 348.693,A -85,B 0,C 180,E1 -17063.614,E2 -17063.614} C_VEL
LIN {X 0,Y 284.299,Z 348.696,A -85,B 0,C 180,E1 -17067.19,E2 -17067.19} C_VEL
LIN {X 0,Y 284.306,Z 348.662,A -85,B 0,C 180,E1 -17070.37,E2 -17070.37} C_VEL
LIN {X 0,Y 284.297,Z 348.696,A -85,B 0,C 180,E1 -17073.579,E2 -17073.579} C_VEL
LIN {X 0,Y 284.32,Z 348.692,A -85,B 0,C 180,E1 -17076.703,E2 -17076.703} C_VEL
LIN {X 0,Y 284.369,Z 348.679,A -85,B 0,C 180,E1 -17079.904,E2 -17079.904} C_VEL
LIN {X 0,Y 284.439,Z 348.671,A -85,B 0,C 180,E1 -17084.492,E2 -17084.492} C_VEL
LIN {X 0,Y 284.455,Z 348.665,A -85,B 0,C 180,E1 -17088.601,E2 -17088.601} C_VEL
LIN {X 0,Y 284.599,Z 348.656,A -85,B 0,C 180,E1 -17091.48,E2 -17091.48} C_VEL
LIN {X 0,Y 284.558,Z 348.661,A -85,B 0,C 180,E1 -17094.331,E2 -17094.331} C_VEL
LIN {X 0,Y 284.836,Z 348.62,A -85,B 0,C 180,E1 -17098.587,E2 -17098.587} C_VEL
LIN {X 0,Y 284.83,Z 348.625,A -85,B 0,C 180,E1 -17101.414,E2 -17101.414} C_VEL
LIN {X 0,Y 284.644,Z 348.643,A -85,B 0,C 180,E1 -17107.092,E2 -17107.092} C_VEL
LIN {X 0,Y 284.506,Z 348.67,A -85,B 0,C 180,E1 -17109.958,E2 -17109.958} C_VEL
LIN {X 0,Y 284.456,Z 348.677,A -85,B 0,C 180,E1 -17114.305,E2 -17114.305} C_VEL
LIN {X 0,Y 284.327,Z 348.695,A -85,B 0,C 180,E1 -17118.744,E2 -17118.744} C_VEL
LIN {X 0,Y 284.327,Z 348.691,A -85,B 0,C 180,E1 -17123.297,E2 -17123.297} C_VEL
LIN {X 0,Y 284.39,Z 348.681,A -85,B 0,C 180,E1 -17127.174,E2 -17127.174} C_VEL
LIN {X 0,Y 284.289,Z 348.69,A -85,B 0,C 180,E1 -17131.276,E2 -17131.276} C_VEL
LIN {X 0,Y 284.338,Z 348.688,A -85,B 0,C 180,E1 -17135.349,E2 -17135.349} C_VEL
LIN {X 0,Y 284.309,Z 348.691,A -85,B 0,C 180,E1 -17138.17,E2 -17138.17} C_VEL
LIN {X 0,Y 284.267,Z 348.697,A -85,B 0,C 180,E1 -17142.126,E2 -17142.126} C_VEL
LIN {X 0,Y 284.246,Z 348.788,A -85,B 0,C 180,E1 -17145.372,E2 -17145.372} C_VEL
LIN {X 0,Y 285.054,Z 351.382,A -85,B 0,C 180,E1 -17146.403,E2 -17146.403} C_VEL
LIN {X 0,Y 287.374,Z 355.209,A -85,B 0,C 180,E1 -17146.918,E2 -17146.918} C_VEL
LIN {X 0,Y 297.169,Z 372.177,A -85,B 0,C 180,E1 -17148.99,E2 -17148.99} C_VEL
LIN {X 0,Y 304.901,Z 387.625,A -85,B 0,C 180,E1 -17150.551,E2 -17150.551} C_VEL
LIN {X 0,Y 310.076,Z 399.272,A -85,B 0,C 180,E1 -17151.572,E2 -17151.572} C_VEL
LIN {X 0,Y 306.631,Z 487.704,A -85,B 0,C 180,E1 -17153.627,E2 -17153.627} C_VEL
LIN {X 0,Y 305.496,Z 502.304,A -85,B 0,C 180,E1 -17154.235,E2 -17154.235} C_VEL
LIN {X 0,Y 303.863,Z 516.271,A -85,B 0,C 180,E1 -17155.081,E2 -17155.081} C_VEL
LIN {X 0,Y 301.769,Z 530.157,A -85,B 0,C 180,E1 -17156.219,E2 -17156.219} C_VEL
LIN {X 0,Y 299.415,Z 542.924,A -85,B 0,C 180,E1 -17157.575,E2 -17157.575} C_VEL
LIN {X 0,Y 296.668,Z 555.015,A -85,B 0,C 180,E1 -17159.184,E2 -17159.184} C_VEL
LIN {X 0,Y 294.095,Z 566.126,A -85,B 0,C 180,E1 -17161.059,E2 -17161.059} C_VEL
LIN {X 0,Y 291.649,Z 575.841,A -85,B 0,C 180,E1 -17163.077,E2 -17163.077} C_VEL
LIN {X 0,Y 289.426,Z 584.315,A -85,B 0,C 180,E1 -17165.237,E2 -17165.237} C_VEL
LIN {X 0,Y 287.252,Z 592.162,A -85,B 0,C 180,E1 -17167.715,E2 -17167.715} C_VEL
LIN {X 0,Y 285.769,Z 597.623,A -85,B 0,C 180,E1 -17169.861,E2 -17169.861} C_VEL
LIN {X 0,Y 284.254,Z 603.334,A -85,B 0,C 180,E1 -17172.741,E2 -17172.741} C_VEL
LIN {X 0,Y 283.254,Z 607.454,A -85,B 0,C 180,E1 -17175.634,E2 -17175.634} C_VEL
LIN {X 0,Y 282.54,Z 610.118,A -85,B 0,C 180,E1 -17178.522,E2 -17178.522} C_VEL
LIN {X 0,Y 282.327,Z 611.399,A -85,B 0,C 180,E1 -17181.41,E2 -17181.41} C_VEL
LIN {X 0,Y 282.382,Z 611.338,A -85,B 0,C 180,E1 -17184.287,E2 -17184.287} C_VEL
LIN {X 0,Y 282.428,Z 609.958,A -85,B 0,C 180,E1 -17187.147,E2 -17187.147} C_VEL
LIN {X 0,Y 282.542,Z 607.243,A -85,B 0,C 180,E1 -17190,E2 -17190} C_VEL
LIN {X 0,Y 283.025,Z 603.112,A -85,B 0,C 180,E1 -17192.847,E2 -17192.847} C_VEL
LIN {X 0,Y 283.783,Z 599.031,A -85,B 0,C 180,E1 -17194.972,E2 -17194.972} C_VEL
LIN {X 0,Y 284.517,Z 593.972,A -85,B 0,C 180,E1 -17197.094,E2 -17197.094} C_VEL
LIN {X 0,Y 286.065,Z 586.724,A -85,B 0,C 180,E1 -17199.545,E2 -17199.545} C_VEL
LIN {X 0,Y 287.727,Z 578.253,A -85,B 0,C 180,E1 -17201.859,E2 -17201.859} C_VEL
LIN {X 0,Y 289.497,Z 568.367,A -85,B 0,C 180,E1 -17204.049,E2 -17204.049} C_VEL
LIN {X 0,Y 291.45,Z 557.97,A -85,B 0,C 180,E1 -17205.92,E2 -17205.92} C_VEL
LIN {X 0,Y 293.47,Z 546.49,A -85,B 0,C 180,E1 -17207.598,E2 -17207.598} C_VEL
LIN {X 0,Y 295.147,Z 535.337,A -85,B 0,C 180,E1 -17208.931,E2 -17208.931} C_VEL
LIN {X 0,Y 296.819,Z 523.305,A -85,B 0,C 180,E1 -17210.079,E2 -17210.079} C_VEL
LIN {X 0,Y 298.289,Z 510.083,A -85,B 0,C 180,E1 -17211.057,E2 -17211.057} C_VEL
LIN {X 0,Y 299.411,Z 496.591,A -85,B 0,C 180,E1 -17211.787,E2 -17211.787} C_VEL
LIN {X 0,Y 300.141,Z 483.043,A -85,B 0,C 180,E1 -17212.274,E2 -17212.274} C_VEL
LIN {X 0,Y 302.757,Z 391.771,A -85,B 0,C 180,E1 -17214.43,E2 -17214.43} C_VEL
LIN {X 0,Y 294.787,Z 371.795,A -85,B 0,C 180,E1 -17215.807,E2 -17215.807} C_VEL
LIN {X 0,Y 287.524,Z 356.209,A -85,B 0,C 180,E1 -17217.071,E2 -17217.071} C_VEL
LIN {X 0,Y 284.827,Z 350.45,A -85,B 0,C 180,E1 -17217.575,E2 -17217.575} C_VEL
LIN {X 0,Y 284.366,Z 348.683,A -85,B 0,C 180,E1 -17218.307,E2 -17218.307} C_VEL
LIN {X 0,Y 284.307,Z 348.694,A -85,B 0,C 180,E1 -17222.944,E2 -17222.944} C_VEL
LIN {X 0,Y 284.35,Z 348.682,A -85,B 0,C 180,E1 -17226.382,E2 -17226.382} C_VEL
LIN {X 0,Y 284.306,Z 348.676,A -85,B 0,C 180,E1 -17229.993,E2 -17229.993} C_VEL
LIN {X 0,Y 284.244,Z 348.699,A -85,B 0,C 180,E1 -17234.189,E2 -17234.189} C_VEL
LIN {X 0,Y 284.269,Z 348.692,A -85,B 0,C 180,E1 -17238.123,E2 -17238.123} C_VEL
LIN {X 0,Y 284.249,Z 348.694,A -85,B 0,C 180,E1 -17239.15,E2 -17239.15} C_VEL
LIN {X 0,Y 283.61,Z 348.783,A -85,B 0,C 180,E1 -17240.332,E2 -17240.332} C_VEL
LIN {X 0,Y 280.77,Z 349.134,A -85,B 0,C 180,E1 -17242.258,E2 -17242.258} C_VEL
LIN {X 0,Y 278.346,Z 349.438,A -85,B 0,C 180,E1 -17243.822,E2 -17243.822} C_VEL
LIN {X 0,Y 277.308,Z 349.568,A -85,B 0,C 180,E1 -17245.035,E2 -17245.035} C_VEL
LIN {X 0,Y 277.226,Z 349.569,A -85,B 0,C 180,E1 -17245.446,E2 -17245.446} C_VEL
LIN {X 0,Y 277.257,Z 349.573,A -85,B 0,C 180,E1 -17249.537,E2 -17249.537} C_VEL
LIN {X 0,Y 277.335,Z 349.545,A -85,B 0,C 180,E1 -17252.861,E2 -17252.861} C_VEL
LIN {X 0,Y 277.285,Z 349.569,A -85,B 0,C 180,E1 -17256.075,E2 -17256.075} C_VEL
LIN {X 0,Y 277.278,Z 349.553,A -85,B 0,C 180,E1 -17260.761,E2 -17260.761} C_VEL
LIN {X 0,Y 277.401,Z 349.546,A -85,B 0,C 180,E1 -17265.324,E2 -17265.324} C_VEL
LIN {X 0,Y 277.447,Z 349.544,A -85,B 0,C 180,E1 -17269.786,E2 -17269.786} C_VEL
LIN {X 0,Y 277.606,Z 349.525,A -85,B 0,C 180,E1 -17272.727,E2 -17272.727} C_VEL
LIN {X 0,Y 277.796,Z 349.503,A -85,B 0,C 180,E1 -17278.55,E2 -17278.55} C_VEL
LIN {X 0,Y 277.795,Z 349.5,A -85,B 0,C 180,E1 -17281.449,E2 -17281.449} C_VEL
LIN {X 0,Y 277.59,Z 349.529,A -85,B 0,C 180,E1 -17287.272,E2 -17287.272} C_VEL
LIN {X 0,Y 277.446,Z 349.536,A -85,B 0,C 180,E1 -17290.213,E2 -17290.213} C_VEL
LIN {X 0,Y 277.401,Z 349.545,A -85,B 0,C 180,E1 -17294.676,E2 -17294.676} C_VEL
LIN {X 0,Y 277.316,Z 349.563,A -85,B 0,C 180,E1 -17299.235,E2 -17299.235} C_VEL
LIN {X 0,Y 277.277,Z 349.571,A -85,B 0,C 180,E1 -17303.925,E2 -17303.925} C_VEL
LIN {X 0,Y 277.262,Z 349.568,A -85,B 0,C 180,E1 -17307.483,E2 -17307.483} C_VEL
LIN {X 0,Y 277.241,Z 349.567,A -85,B 0,C 180,E1 -17310.473,E2 -17310.473} C_VEL
LIN {X 0,Y 277.24,Z 349.571,A -85,B 0,C 180,E1 -17313.896,E2 -17313.896} C_VEL
LIN {X 0,Y 277.261,Z 349.569,A -85,B 0,C 180,E1 -17317.47,E2 -17317.47} C_VEL
LIN {X 0,Y 277.204,Z 349.564,A -85,B 0,C 180,E1 -17321.237,E2 -17321.237} C_VEL
LIN {X 0,Y 277.196,Z 349.579,A -85,B 0,C 180,E1 -17325.227,E2 -17325.227} C_VEL
LIN {X 0,Y 277.218,Z 349.583,A -85,B 0,C 180,E1 -17329.513,E2 -17329.513} C_VEL
LIN {X 0,Y 277.272,Z 349.764,A -85,B 0,C 180,E1 -17331.203,E2 -17331.203} C_VEL
LIN {X 0,Y 279.609,Z 358.835,A -85,B 0,C 180,E1 -17334.362,E2 -17334.362} C_VEL
LIN {X 0,Y 280.763,Z 363.736,A -85,B 0,C 180,E1 -17335.965,E2 -17335.965} C_VEL
LIN {X 0,Y 289.339,Z 383.321,A -85,B 0,C 180,E1 -17337.543,E2 -17337.543} C_VEL
LIN {X 0,Y 292.498,Z 391.509,A -85,B 0,C 180,E1 -17338.122,E2 -17338.122} C_VEL
LIN {X 0,Y 295.981,Z 414.954,A -85,B 0,C 180,E1 -17339.132,E2 -17339.132} C_VEL
LIN {X 0,Y 293.156,Z 502.536,A -85,B 0,C 180,E1 -17341.252,E2 -17341.252} C_VEL
LIN {X 0,Y 292.102,Z 516.27,A -85,B 0,C 180,E1 -17341.825,E2 -17341.825} C_VEL
LIN {X 0,Y 290.647,Z 529.823,A -85,B 0,C 180,E1 -17342.651,E2 -17342.651} C_VEL
LIN {X 0,Y 289.032,Z 542.157,A -85,B 0,C 180,E1 -17343.657,E2 -17343.657} C_VEL
LIN {X 0,Y 287.103,Z 554.84,A -85,B 0,C 180,E1 -17344.988,E2 -17344.988} C_VEL
LIN {X 0,Y 285.254,Z 565.674,A -85,B 0,C 180,E1 -17346.4,E2 -17346.4} C_VEL
LIN {X 0,Y 283.086,Z 576.62,A -85,B 0,C 180,E1 -17348.137,E2 -17348.137} C_VEL
LIN {X 0,Y 280.964,Z 587.44,A -85,B 0,C 180,E1 -17350.265,E2 -17350.265} C_VEL
LIN {X 0,Y 279.26,Z 596.369,A -85,B 0,C 180,E1 -17352.423,E2 -17352.423} C_VEL
LIN {X 0,Y 278.029,Z 603.796,A -85,B 0,C 180,E1 -17354.609,E2 -17354.609} C_VEL
LIN {X 0,Y 276.891,Z 609.967,A -85,B 0,C 180,E1 -17356.795,E2 -17356.795} C_VEL
LIN {X 0,Y 276.054,Z 615.075,A -85,B 0,C 180,E1 -17358.993,E2 -17358.993} C_VEL
LIN {X 0,Y 275.518,Z 620.333,A -85,B 0,C 180,E1 -17361.935,E2 -17361.935} C_VEL
LIN {X 0,Y 275.319,Z 623.768,A -85,B 0,C 180,E1 -17364.587,E2 -17364.587} C_VEL
LIN {X 0,Y 275.256,Z 625.939,A -85,B 0,C 180,E1 -17367.073,E2 -17367.073} C_VEL
LIN {X 0,Y 275.277,Z 627.208,A -85,B 0,C 180,E1 -17370,E2 -17370} C_VEL
LIN {X 0,Y 275.24,Z 627.126,A -85,B 0,C 180,E1 -17372.927,E2 -17372.927} C_VEL
LIN {X 0,Y 275.295,Z 625.711,A -85,B 0,C 180,E1 -17375.861,E2 -17375.861} C_VEL
LIN {X 0,Y 275.672,Z 622.941,A -85,B 0,C 180,E1 -17378.799,E2 -17378.799} C_VEL
LIN {X 0,Y 276.426,Z 618.744,A -85,B 0,C 180,E1 -17381.735,E2 -17381.735} C_VEL
LIN {X 0,Y 277.933,Z 613.005,A -85,B 0,C 180,E1 -17384.647,E2 -17384.647} C_VEL
LIN {X 0,Y 279.452,Z 606.726,A -85,B 0,C 180,E1 -17387.124,E2 -17387.124} C_VEL
LIN {X 0,Y 281.712,Z 598.575,A -85,B 0,C 180,E1 -17389.681,E2 -17389.681} C_VEL
LIN {X 0,Y 284.031,Z 590.243,A -85,B 0,C 180,E1 -17391.786,E2 -17391.786} C_VEL
LIN {X 0,Y 286.754,Z 580.232,A -85,B 0,C 180,E1 -17393.853,E2 -17393.853} C_VEL
LIN {X 0,Y 289.591,Z 569.092,A -85,B 0,C 180,E1 -17395.708,E2 -17395.708} C_VEL
LIN {X 0,Y 292.388,Z 556.622,A -85,B 0,C 180,E1 -17397.367,E2 -17397.367} C_VEL
LIN {X 0,Y 294.738,Z 544.282,A -85,B 0,C 180,E1 -17398.677,E2 -17398.677} C_VEL
LIN {X 0,Y 296.895,Z 531.644,A -85,B 0,C 180,E1 -17399.71,E2 -17399.71} C_VEL
LIN {X 0,Y 298.852,Z 517.476,A -85,B 0,C 180,E1 -17400.566,E2 -17400.566} C_VEL
LIN {X 0,Y 300.165,Z 503.583,A -85,B 0,C 180,E1 -17401.149,E2 -17401.149} C_VEL
LIN {X 0,Y 301.266,Z 478.165,A -85,B 0,C 180,E1 -17401.796,E2 -17401.796} C_VEL
LIN {X 0,Y 303.527,Z 417.022,A -85,B 0,C 180,E1 -17403.233,E2 -17403.233} C_VEL
LIN {X 0,Y 301.047,Z 402.889,A -85,B 0,C 180,E1 -17403.98,E2 -17403.98} C_VEL
LIN {X 0,Y 294.083,Z 387.734,A -85,B 0,C 180,E1 -17405.442,E2 -17405.442} C_VEL
LIN {X 0,Y 287.456,Z 374.634,A -85,B 0,C 180,E1 -17406.888,E2 -17406.888} C_VEL
LIN {X 0,Y 283.016,Z 366.581,A -85,B 0,C 180,E1 -17407.889,E2 -17407.889} C_VEL
LIN {X 0,Y 281.088,Z 362.922,A -85,B 0,C 180,E1 -17408.371,E2 -17408.371} C_VEL
LIN {X 0,Y 278.545,Z 354.095,A -85,B 0,C 180,E1 -17411.9,E2 -17411.9} C_VEL
LIN {X 0,Y 277.209,Z 349.572,A -85,B 0,C 180,E1 -17413.901,E2 -17413.901} C_VEL
LIN {X 0,Y 277.21,Z 349.573,A -85,B 0,C 180,E1 -17417.325,E2 -17417.325} C_VEL
LIN {X 0,Y 277.259,Z 349.571,A -85,B 0,C 180,E1 -17421.792,E2 -17421.792} C_VEL
LIN {X 0,Y 277.278,Z 349.568,A -85,B 0,C 180,E1 -17424.341,E2 -17424.341} C_VEL
LIN {X 0,Y 277.23,Z 349.567,A -85,B 0,C 180,E1 -17427.835,E2 -17427.835} C_VEL
LIN {X 0,Y 277.259,Z 349.565,A -85,B 0,C 180,E1 -17432.518,E2 -17432.518} C_VEL
LIN {X 0,Y 277.274,Z 349.564,A -85,B 0,C 180,E1 -17436.075,E2 -17436.075} C_VEL
LIN {X 0,Y 277.316,Z 349.564,A -85,B 0,C 180,E1 -17440.765,E2 -17440.765} C_VEL
LIN {X 0,Y 277.4,Z 349.553,A -85,B 0,C 180,E1 -17445.324,E2 -17445.324} C_VEL
LIN {X 0,Y 277.446,Z 349.547,A -85,B 0,C 180,E1 -17449.787,E2 -17449.787} C_VEL
LIN {X 0,Y 277.591,Z 349.52,A -85,B 0,C 180,E1 -17452.728,E2 -17452.728} C_VEL
LIN {X 0,Y 277.802,Z 349.496,A -85,B 0,C 180,E1 -17458.551,E2 -17458.551} C_VEL
LIN {X 0,Y 277.797,Z 349.5,A -85,B 0,C 180,E1 -17461.45,E2 -17461.45} C_VEL
LIN {X 0,Y 277.602,Z 349.519,A -85,B 0,C 180,E1 -17467.273,E2 -17467.273} C_VEL
LIN {X 0,Y 277.447,Z 349.549,A -85,B 0,C 180,E1 -17470.214,E2 -17470.214} C_VEL
LIN {X 0,Y 277.402,Z 349.557,A -85,B 0,C 180,E1 -17474.676,E2 -17474.676} C_VEL
LIN {X 0,Y 277.279,Z 349.569,A -85,B 0,C 180,E1 -17479.239,E2 -17479.239} C_VEL
LIN {X 0,Y 277.291,Z 349.564,A -85,B 0,C 180,E1 -17483.925,E2 -17483.925} C_VEL
LIN {X 0,Y 277.319,Z 349.56,A -85,B 0,C 180,E1 -17487.505,E2 -17487.505} C_VEL
LIN {X 0,Y 277.268,Z 349.569,A -85,B 0,C 180,E1 -17490.483,E2 -17490.483} C_VEL
LIN {X 0,Y 277.243,Z 349.57,A -85,B 0,C 180,E1 -17493.897,E2 -17493.897} C_VEL
LIN {X 0,Y 277.264,Z 349.565,A -85,B 0,C 180,E1 -17497.471,E2 -17497.471} C_VEL
LIN {X 0,Y 277.207,Z 349.581,A -85,B 0,C 180,E1 -17501.238,E2 -17501.238} C_VEL
LIN {X 0,Y 277.213,Z 349.711,A -85,B 0,C 180,E1 -17504.345,E2 -17504.345} C_VEL
LIN {X 0,Y 277.754,Z 351.545,A -85,B 0,C 180,E1 -17505.113,E2 -17505.113} C_VEL
LIN {X 0,Y 280.21,Z 355.566,A -85,B 0,C 180,E1 -17505.693,E2 -17505.693} C_VEL
LIN {X 0,Y 286.664,Z 366.354,A -85,B 0,C 180,E1 -17507.156,E2 -17507.156} C_VEL
LIN {X 0,Y 294.436,Z 380.424,A -85,B 0,C 180,E1 -17508.827,E2 -17508.827} C_VEL
LIN {X 0,Y 300.569,Z 393.085,A -85,B 0,C 180,E1 -17510.104,E2 -17510.104} C_VEL
LIN {X 0,Y 304.187,Z 401.355,A -85,B 0,C 180,E1 -17510.846,E2 -17510.846} C_VEL
LIN {X 0,Y 300.7,Z 487.959,A -85,B 0,C 180,E1 -17512.895,E2 -17512.895} C_VEL
LIN {X 0,Y 299.534,Z 502.544,A -85,B 0,C 180,E1 -17513.514,E2 -17513.514} C_VEL
LIN {X 0,Y 297.836,Z 516.5,A -85,B 0,C 180,E1 -17514.371,E2 -17514.371} C_VEL
LIN {X 0,Y 295.826,Z 529.487,A -85,B 0,C 180,E1 -17515.446,E2 -17515.446} C_VEL
LIN {X 0,Y 293.712,Z 540.624,A -85,B 0,C 180,E1 -17516.61,E2 -17516.61} C_VEL
LIN {X 0,Y 291.117,Z 552.329,A -85,B 0,C 180,E1 -17518.124,E2 -17518.124} C_VEL
LIN {X 0,Y 288.709,Z 562.04,A -85,B 0,C 180,E1 -17519.662,E2 -17519.662} C_VEL
LIN {X 0,Y 286.371,Z 571.145,A -85,B 0,C 180,E1 -17521.409,E2 -17521.409} C_VEL
LIN {X 0,Y 284.061,Z 580.261,A -85,B 0,C 180,E1 -17523.556,E2 -17523.556} C_VEL
LIN {X 0,Y 281.461,Z 588.94,A -85,B 0,C 180,E1 -17526.062,E2 -17526.062} C_VEL
LIN {X 0,Y 279.408,Z 596.126,A -85,B 0,C 180,E1 -17528.701,E2 -17528.701} C_VEL
LIN {X 0,Y 277.692,Z 602.133,A -85,B 0,C 180,E1 -17531.558,E2 -17531.558} C_VEL
LIN {X 0,Y 276.745,Z 605.655,A -85,B 0,C 180,E1 -17533.779,E2 -17533.779} C_VEL
LIN {X 0,Y 275.825,Z 609.075,A -85,B 0,C 180,E1 -17536.743,E2 -17536.743} C_VEL
LIN {X 0,Y 275.302,Z 611.085,A -85,B 0,C 180,E1 -17539.706,E2 -17539.706} C_VEL
LIN {X 0,Y 275.229,Z 611.74,A -85,B 0,C 180,E1 -17542.665,E2 -17542.665} C_VEL
LIN {X 0,Y 275.333,Z 611.427,A -85,B 0,C 180,E1 -17544.567,E2 -17544.567} C_VEL
LIN {X 0,Y 275.332,Z 610.23,A -85,B 0,C 180,E1 -17547.074,E2 -17547.074} C_VEL
LIN {X 0,Y 275.454,Z 607.555,A -85,B 0,C 180,E1 -17550,E2 -17550} C_VEL
LIN {X 0,Y 275.944,Z 603.467,A -85,B 0,C 180,E1 -17552.92,E2 -17552.92} C_VEL
LIN {X 0,Y 276.731,Z 599.426,A -85,B 0,C 180,E1 -17555.099,E2 -17555.099} C_VEL
LIN {X 0,Y 277.495,Z 594.396,A -85,B 0,C 180,E1 -17557.275,E2 -17557.275} C_VEL
LIN {X 0,Y 279.093,Z 587.199,A -85,B 0,C 180,E1 -17559.786,E2 -17559.786} C_VEL
LIN {X 0,Y 280.767,Z 578.97,A -85,B 0,C 180,E1 -17562.11,E2 -17562.11} C_VEL
LIN {X 0,Y 282.325,Z 570.82,A -85,B 0,C 180,E1 -17564.009,E2 -17564.009} C_VEL
LIN {X 0,Y 284.086,Z 561.678,A -85,B 0,C 180,E1 -17565.791,E2 -17565.791} C_VEL
LIN {X 0,Y 286.109,Z 550.961,A -85,B 0,C 180,E1 -17567.512,E2 -17567.512} C_VEL
LIN {X 0,Y 288.035,Z 539.255,A -85,B 0,C 180,E1 -17569.047,E2 -17569.047} C_VEL
LIN {X 0,Y 289.94,Z 526.34,A -85,B 0,C 180,E1 -17570.391,E2 -17570.391} C_VEL
LIN {X 0,Y 291.447,Z 513.976,A -85,B 0,C 180,E1 -17571.39,E2 -17571.39} C_VEL
LIN {X 0,Y 292.75,Z 500.312,A -85,B 0,C 180,E1 -17572.216,E2 -17572.216} C_VEL
LIN {X 0,Y 293.626,Z 486.162,A -85,B 0,C 180,E1 -17572.795,E2 -17572.795} C_VEL
LIN {X 0,Y 296.464,Z 393.456,A -85,B 0,C 180,E1 -17575.035,E2 -17575.035} C_VEL
LIN {X 0,Y 287.8,Z 372.036,A -85,B 0,C 180,E1 -17576.589,E2 -17576.589} C_VEL
LIN {X 0,Y 280.593,Z 356.861,A -85,B 0,C 180,E1 -17577.895,E2 -17577.895} C_VEL
LIN {X 0,Y 277.567,Z 350.677,A -85,B 0,C 180,E1 -17578.481,E2 -17578.481} C_VEL
LIN {X 0,Y 277.308,Z 349.561,A -85,B 0,C 180,E1 -17578.992,E2 -17578.992} C_VEL
LIN {X 0,Y 277.256,Z 349.573,A -85,B 0,C 180,E1 -17583.227,E2 -17583.227} C_VEL
LIN {X 0,Y 277.325,Z 349.554,A -85,B 0,C 180,E1 -17585.81,E2 -17585.81} C_VEL
LIN {X 0,Y 277.238,Z 349.561,A -85,B 0,C 180,E1 -17589.326,E2 -17589.326} C_VEL
LIN {X 0,Y 277.208,Z 349.58,A -85,B 0,C 180,E1 -17593.197,E2 -17593.197} C_VEL
LIN {X 0,Y 277.212,Z 349.577,A -85,B 0,C 180,E1 -17597.324,E2 -17597.324} C_VEL
LIN {X 0,Y 277.258,Z 349.565,A -85,B 0,C 180,E1 -17601.792,E2 -17601.792} C_VEL
LIN {X 0,Y 277.226,Z 349.569,A -85,B 0,C 180,E1 -17605.446,E2 -17605.446} C_VEL
LIN {X 0,Y 276.55,Z 349.655,A -85,B 0,C 180,E1 -17606.658,E2 -17606.658} C_VEL
LIN {X 0,Y 273.662,Z 350.02,A -85,B 0,C 180,E1 -17608.633,E2 -17608.633} C_VEL
LIN {X 0,Y 271.25,Z 350.32,A -85,B 0,C 180,E1 -17610.239,E2 -17610.239} C_VEL
LIN {X 0,Y 270.271,Z 350.429,A -85,B 0,C 180,E1 -17611.484,E2 -17611.484} C_VEL
LIN {X 0,Y 270.222,Z 350.431,A -85,B 0,C 180,E1 -17611.905,E2 -17611.905} C_VEL
LIN {X 0,Y 270.229,Z 350.449,A -85,B 0,C 180,E1 -17615.538,E2 -17615.538} C_VEL
LIN {X 0,Y 270.217,Z 350.428,A -85,B 0,C 180,E1 -17620.237,E2 -17620.237} C_VEL
LIN {X 0,Y 270.361,Z 350.425,A -85,B 0,C 180,E1 -17624.932,E2 -17624.932} C_VEL
LIN {X 0,Y 270.399,Z 350.42,A -85,B 0,C 180,E1 -17629.517,E2 -17629.517} C_VEL
LIN {X 0,Y 270.566,Z 350.404,A -85,B 0,C 180,E1 -17632.537,E2 -17632.537} C_VEL
LIN {X 0,Y 270.761,Z 350.379,A -85,B 0,C 180,E1 -17638.512,E2 -17638.512} C_VEL
LIN {X 0,Y 270.758,Z 350.377,A -85,B 0,C 180,E1 -17641.487,E2 -17641.487} C_VEL
LIN {X 0,Y 270.552,Z 350.406,A -85,B 0,C 180,E1 -17647.462,E2 -17647.462} C_VEL
LIN {X 0,Y 270.379,Z 350.418,A -85,B 0,C 180,E1 -17650.483,E2 -17650.483} C_VEL
LIN {X 0,Y 270.369,Z 350.419,A -85,B 0,C 180,E1 -17655.066,E2 -17655.066} C_VEL
LIN {X 0,Y 270.253,Z 350.44,A -85,B 0,C 180,E1 -17659.759,E2 -17659.759} C_VEL
LIN {X 0,Y 270.218,Z 350.445,A -85,B 0,C 180,E1 -17664.591,E2 -17664.591} C_VEL
LIN {X 0,Y 270.192,Z 350.451,A -85,B 0,C 180,E1 -17667.917,E2 -17667.917} C_VEL
LIN {X 0,Y 270.167,Z 350.452,A -85,B 0,C 180,E1 -17671.35,E2 -17671.35} C_VEL
LIN {X 0,Y 270.195,Z 350.451,A -85,B 0,C 180,E1 -17674.906,E2 -17674.906} C_VEL
LIN {X 0,Y 270.192,Z 350.454,A -85,B 0,C 180,E1 -17678.711,E2 -17678.711} C_VEL
LIN {X 0,Y 270.16,Z 350.455,A -85,B 0,C 180,E1 -17683.25,E2 -17683.25} C_VEL
LIN {X 0,Y 270.167,Z 350.457,A -85,B 0,C 180,E1 -17687.442,E2 -17687.442} C_VEL
LIN {X 0,Y 270.182,Z 350.486,A -85,B 0,C 180,E1 -17690.412,E2 -17690.412} C_VEL
LIN {X 0,Y 272.95,Z 361.188,A -85,B 0,C 180,E1 -17694.262,E2 -17694.262} C_VEL
LIN {X 0,Y 273.458,Z 363.411,A -85,B 0,C 180,E1 -17695.02,E2 -17695.02} C_VEL
LIN {X 0,Y 282.137,Z 382.883,A -85,B 0,C 180,E1 -17696.691,E2 -17696.691} C_VEL
LIN {X 0,Y 286.504,Z 393.911,A -85,B 0,C 180,E1 -17697.519,E2 -17697.519} C_VEL
LIN {X 0,Y 289.698,Z 416.759,A -85,B 0,C 180,E1 -17698.515,E2 -17698.515} C_VEL
LIN {X 0,Y 286.835,Z 501.866,A -85,B 0,C 180,E1 -17700.608,E2 -17700.608} C_VEL
LIN {X 0,Y 285.752,Z 515.756,A -85,B 0,C 180,E1 -17701.191,E2 -17701.191} C_VEL
LIN {X 0,Y 284.167,Z 529.958,A -85,B 0,C 180,E1 -17702.073,E2 -17702.073} C_VEL
LIN {X 0,Y 282.37,Z 543.109,A -85,B 0,C 180,E1 -17703.185,E2 -17703.185} C_VEL
LIN {X 0,Y 280.429,Z 555.348,A -85,B 0,C 180,E1 -17704.518,E2 -17704.518} C_VEL
LIN {X 0,Y 278.48,Z 566.24,A -85,B 0,C 180,E1 -17705.988,E2 -17705.988} C_VEL
LIN {X 0,Y 276.478,Z 576.074,A -85,B 0,C 180,E1 -17707.587,E2 -17707.587} C_VEL
LIN {X 0,Y 274.587,Z 585.305,A -85,B 0,C 180,E1 -17709.395,E2 -17709.395} C_VEL
LIN {X 0,Y 272.688,Z 594.555,A -85,B 0,C 180,E1 -17711.596,E2 -17711.596} C_VEL
LIN {X 0,Y 271.109,Z 603.396,A -85,B 0,C 180,E1 -17714.206,E2 -17714.206} C_VEL
LIN {X 0,Y 269.936,Z 609.606,A -85,B 0,C 180,E1 -17716.449,E2 -17716.449} C_VEL
LIN {X 0,Y 269.028,Z 614.742,A -85,B 0,C 180,E1 -17718.701,E2 -17718.701} C_VEL
LIN {X 0,Y 268.462,Z 620.039,A -85,B 0,C 180,E1 -17721.722,E2 -17721.722} C_VEL
LIN {X 0,Y 268.215,Z 623.742,A -85,B 0,C 180,E1 -17724.689,E2 -17724.689} C_VEL
LIN {X 0,Y 268.168,Z 625.692,A -85,B 0,C 180,E1 -17726.996,E2 -17726.996} C_VEL
LIN {X 0,Y 268.201,Z 626.996,A -85,B 0,C 180,E1 -17730,E2 -17730} C_VEL
LIN {X 0,Y 268.151,Z 626.945,A -85,B 0,C 180,E1 -17733.005,E2 -17733.005} C_VEL
LIN {X 0,Y 268.218,Z 625.557,A -85,B 0,C 180,E1 -17736.016,E2 -17736.016} C_VEL
LIN {X 0,Y 268.632,Z 622.816,A -85,B 0,C 180,E1 -17739.031,E2 -17739.031} C_VEL
LIN {X 0,Y 269.431,Z 618.65,A -85,B 0,C 180,E1 -17742.044,E2 -17742.044} C_VEL
LIN {X 0,Y 271.003,Z 612.944,A -85,B 0,C 180,E1 -17745.03,E2 -17745.03} C_VEL
LIN {X 0,Y 272.505,Z 607.156,A -85,B 0,C 180,E1 -17747.4,E2 -17747.4} C_VEL
LIN {X 0,Y 274.636,Z 599.821,A -85,B 0,C 180,E1 -17749.82,E2 -17749.82} C_VEL
LIN {X 0,Y 276.982,Z 591.786,A -85,B 0,C 180,E1 -17751.978,E2 -17751.978} C_VEL
LIN {X 0,Y 279.798,Z 582.12,A -85,B 0,C 180,E1 -17754.089,E2 -17754.089} C_VEL
LIN {X 0,Y 282.662,Z 571.416,A -85,B 0,C 180,E1 -17755.99,E2 -17755.99} C_VEL
LIN {X 0,Y 285.518,Z 559.311,A -85,B 0,C 180,E1 -17757.727,E2 -17757.727} C_VEL
LIN {X 0,Y 288.191,Z 546.423,A -85,B 0,C 180,E1 -17759.191,E2 -17759.191} C_VEL
LIN {X 0,Y 290.598,Z 533.357,A -85,B 0,C 180,E1 -17760.321,E2 -17760.321} C_VEL
LIN {X 0,Y 292.708,Z 519.098,A -85,B 0,C 180,E1 -17761.229,E2 -17761.229} C_VEL
LIN {X 0,Y 294.147,Z 504.975,A -85,B 0,C 180,E1 -17761.86,E2 -17761.86} C_VEL
LIN {X 0,Y 295.121,Z 487.378,A -85,B 0,C 180,E1 -17762.34,E2 -17762.34} C_VEL
LIN {X 0,Y 297.757,Z 418.122,A -85,B 0,C 180,E1 -17763.998,E2 -17763.998} C_VEL
LIN {X 0,Y 295.611,Z 405.85,A -85,B 0,C 180,E1 -17764.671,E2 -17764.671} C_VEL
LIN {X 0,Y 289.375,Z 392.148,A -85,B 0,C 180,E1 -17766.032,E2 -17766.032} C_VEL
LIN {X 0,Y 282.763,Z 378.892,A -85,B 0,C 180,E1 -17767.532,E2 -17767.532} C_VEL
LIN {X 0,Y 278.171,Z 370.591,A -85,B 0,C 180,E1 -17768.606,E2 -17768.606} C_VEL
LIN {X 0,Y 273.742,Z 362.613,A -85,B 0,C 180,E1 -17769.735,E2 -17769.735} C_VEL
LIN {X 0,Y 271.704,Z 355.614,A -85,B 0,C 180,E1 -17772.665,E2 -17772.665} C_VEL
LIN {X 0,Y 270.161,Z 350.448,A -85,B 0,C 180,E1 -17775.014,E2 -17775.014} C_VEL
LIN {X 0,Y 270.164,Z 350.456,A -85,B 0,C 180,E1 -17778.971,E2 -17778.971} C_VEL
LIN {X 0,Y 270.211,Z 350.45,A -85,B 0,C 180,E1 -17783.258,E2 -17783.258} C_VEL
LIN {X 0,Y 270.195,Z 350.453,A -85,B 0,C 180,E1 -17786.892,E2 -17786.892} C_VEL
LIN {X 0,Y 270.153,Z 350.423,A -85,B 0,C 180,E1 -17790.378,E2 -17790.378} C_VEL
LIN {X 0,Y 270.194,Z 350.454,A -85,B 0,C 180,E1 -17793.757,E2 -17793.757} C_VEL
LIN {X 0,Y 270.193,Z 350.452,A -85,B 0,C 180,E1 -17797.036,E2 -17797.036} C_VEL
LIN {X 0,Y 270.253,Z 350.439,A -85,B 0,C 180,E1 -17800.241,E2 -17800.241} C_VEL
LIN {X 0,Y 270.369,Z 350.427,A -85,B 0,C 180,E1 -17804.934,E2 -17804.934} C_VEL
LIN {X 0,Y 270.379,Z 350.424,A -85,B 0,C 180,E1 -17809.517,E2 -17809.517} C_VEL
LIN {X 0,Y 270.553,Z 350.398,A -85,B 0,C 180,E1 -17812.538,E2 -17812.538} C_VEL
LIN {X 0,Y 270.767,Z 350.371,A -85,B 0,C 180,E1 -17818.513,E2 -17818.513} C_VEL
LIN {X 0,Y 270.763,Z 350.376,A -85,B 0,C 180,E1 -17821.488,E2 -17821.488} C_VEL
LIN {X 0,Y 270.562,Z 350.396,A -85,B 0,C 180,E1 -17827.463,E2 -17827.463} C_VEL
LIN {X 0,Y 270.399,Z 350.428,A -85,B 0,C 180,E1 -17830.483,E2 -17830.483} C_VEL
LIN {X 0,Y 270.361,Z 350.43,A -85,B 0,C 180,E1 -17835.068,E2 -17835.068} C_VEL
LIN {X 0,Y 270.218,Z 350.446,A -85,B 0,C 180,E1 -17839.763,E2 -17839.763} C_VEL
LIN {X 0,Y 270.233,Z 350.441,A -85,B 0,C 180,E1 -17844.59,E2 -17844.59} C_VEL
LIN {X 0,Y 270.266,Z 350.437,A -85,B 0,C 180,E1 -17847.91,E2 -17847.91} C_VEL
LIN {X 0,Y 270.18,Z 350.447,A -85,B 0,C 180,E1 -17851.349,E2 -17851.349} C_VEL
LIN {X 0,Y 270.198,Z 350.446,A -85,B 0,C 180,E1 -17854.907,E2 -17854.907} C_VEL
LIN {X 0,Y 270.195,Z 350.454,A -85,B 0,C 180,E1 -17858.712,E2 -17858.712} C_VEL
LIN {X 0,Y 270.182,Z 350.502,A -85,B 0,C 180,E1 -17863.193,E2 -17863.193} C_VEL
LIN {X 0,Y 270.441,Z 351.712,A -85,B 0,C 180,E1 -17863.72,E2 -17863.72} C_VEL
LIN {X 0,Y 272.048,Z 354.513,A -85,B 0,C 180,E1 -17864.136,E2 -17864.136} C_VEL
LIN {X 0,Y 274.313,Z 357.966,A -85,B 0,C 180,E1 -17864.691,E2 -17864.691} C_VEL
LIN {X 0,Y 279.56,Z 366.435,A -85,B 0,C 180,E1 -17865.94,E2 -17865.94} C_VEL
LIN {X 0,Y 287.641,Z 380.741,A -85,B 0,C 180,E1 -17867.772,E2 -17867.772} C_VEL
LIN {X 0,Y 294.851,Z 395.373,A -85,B 0,C 180,E1 -17869.341,E2 -17869.341} C_VEL
LIN {X 0,Y 298.356,Z 403.375,A -85,B 0,C 180,E1 -17870.09,E2 -17870.09} C_VEL
LIN {X 0,Y 294.85,Z 487.952,A -85,B 0,C 180,E1 -17872.125,E2 -17872.125} C_VEL
LIN {X 0,Y 293.625,Z 502.532,A -85,B 0,C 180,E1 -17872.746,E2 -17872.746} C_VEL
LIN {X 0,Y 291.853,Z 516.733,A -85,B 0,C 180,E1 -17873.632,E2 -17873.632} C_VEL
LIN {X 0,Y 289.595,Z 530.603,A -85,B 0,C 180,E1 -17874.805,E2 -17874.805} C_VEL
LIN {X 0,Y 287.004,Z 543.592,A -85,B 0,C 180,E1 -17876.233,E2 -17876.233} C_VEL
LIN {X 0,Y 284.124,Z 555.444,A -85,B 0,C 180,E1 -17877.873,E2 -17877.873} C_VEL
LIN {X 0,Y 281.518,Z 565.65,A -85,B 0,C 180,E1 -17879.634,E2 -17879.634} C_VEL
LIN {X 0,Y 278.773,Z 575.619,A -85,B 0,C 180,E1 -17881.755,E2 -17881.755} C_VEL
LIN {X 0,Y 276.403,Z 584.113,A -85,B 0,C 180,E1 -17883.986,E2 -17883.986} C_VEL
LIN {X 0,Y 274.205,Z 591.058,A -85,B 0,C 180,E1 -17886.192,E2 -17886.192} C_VEL
LIN {X 0,Y 272.19,Z 597.63,A -85,B 0,C 180,E1 -17888.809,E2 -17888.809} C_VEL
LIN {X 0,Y 270.46,Z 603.433,A -85,B 0,C 180,E1 -17891.831,E2 -17891.831} C_VEL
LIN {X 0,Y 269.267,Z 607.739,A -85,B 0,C 180,E1 -17894.957,E2 -17894.957} C_VEL
LIN {X 0,Y 268.47,Z 610.385,A -85,B 0,C 180,E1 -17897.912,E2 -17897.912} C_VEL
LIN {X 0,Y 268.16,Z 611.754,A -85,B 0,C 180,E1 -17900.953,E2 -17900.953} C_VEL
LIN {X 0,Y 268.186,Z 611.788,A -85,B 0,C 180,E1 -17903.983,E2 -17903.983} C_VEL
LIN {X 0,Y 268.238,Z 610.498,A -85,B 0,C 180,E1 -17906.996,E2 -17906.996} C_VEL
LIN {X 0,Y 268.369,Z 607.865,A -85,B 0,C 180,E1 -17910,E2 -17910} C_VEL
LIN {X 0,Y 268.866,Z 603.82,A -85,B 0,C 180,E1 -17912.997,E2 -17912.997} C_VEL
LIN {X 0,Y 269.664,Z 599.81,A -85,B 0,C 180,E1 -17915.233,E2 -17915.233} C_VEL
LIN {X 0,Y 270.478,Z 594.817,A -85,B 0,C 180,E1 -17917.465,E2 -17917.465} C_VEL
LIN {X 0,Y 272.109,Z 587.672,A -85,B 0,C 180,E1 -17920.04,E2 -17920.04} C_VEL
LIN {X 0,Y 273.794,Z 579.857,A -85,B 0,C 180,E1 -17922.323,E2 -17922.323} C_VEL
LIN {X 0,Y 275.466,Z 571.415,A -85,B 0,C 180,E1 -17924.366,E2 -17924.366} C_VEL
LIN {X 0,Y 277.71,Z 560.415,A -85,B 0,C 180,E1 -17926.541,E2 -17926.541} C_VEL
LIN {X 0,Y 279.848,Z 549.397,A -85,B 0,C 180,E1 -17928.295,E2 -17928.295} C_VEL
LIN {X 0,Y 281.845,Z 537.27,A -85,B 0,C 180,E1 -17929.861,E2 -17929.861} C_VEL
LIN {X 0,Y 283.625,Z 525.619,A -85,B 0,C 180,E1 -17931.056,E2 -17931.056} C_VEL
LIN {X 0,Y 285.146,Z 513.002,A -85,B 0,C 180,E1 -17932.077,E2 -17932.077} C_VEL
LIN {X 0,Y 286.563,Z 498.708,A -85,B 0,C 180,E1 -17932.913,E2 -17932.913} C_VEL
LIN {X 0,Y 287.384,Z 484.789,A -85,B 0,C 180,E1 -17933.462,E2 -17933.462} C_VEL
LIN {X 0,Y 290.216,Z 395.208,A -85,B 0,C 180,E1 -17935.664,E2 -17935.664} C_VEL
LIN {X 0,Y 282.275,Z 375.581,A -85,B 0,C 180,E1 -17937.141,E2 -17937.141} C_VEL
LIN {X 0,Y 275.32,Z 360.761,A -85,B 0,C 180,E1 -17938.453,E2 -17938.453} C_VEL
LIN {X 0,Y 271.413,Z 353.488,A -85,B 0,C 180,E1 -17939.195,E2 -17939.195} C_VEL
LIN {X 0,Y 270.33,Z 350.784,A -85,B 0,C 180,E1 -17939.483,E2 -17939.483} C_VEL
LIN {X 0,Y 270.251,Z 350.444,A -85,B 0,C 180,E1 -17939.809,E2 -17939.809} C_VEL
LIN {X 0,Y 270.221,Z 350.452,A -85,B 0,C 180,E1 -17943.666,E2 -17943.666} C_VEL
LIN {X 0,Y 270.238,Z 350.442,A -85,B 0,C 180,E1 -17946.736,E2 -17946.736} C_VEL
LIN {X 0,Y 270.173,Z 350.435,A -85,B 0,C 180,E1 -17950.565,E2 -17950.565} C_VEL
LIN {X 0,Y 270.151,Z 350.454,A -85,B 0,C 180,E1 -17954.619,E2 -17954.619} C_VEL
LIN {X 0,Y 270.166,Z 350.45,A -85,B 0,C 180,E1 -17958.971,E2 -17958.971} C_VEL
LIN {X 0,Y 270.212,Z 350.446,A -85,B 0,C 180,E1 -17963.257,E2 -17963.257} C_VEL
LIN {X 0,Y 270.198,Z 350.444,A -85,B 0,C 180,E1 -17966.891,E2 -17966.891} C_VEL
LIN {X 0,Y 270.188,Z 350.452,A -85,B 0,C 180,E1 -17970.381,E2 -17970.381} C_VEL
LIN {X 0,Y 270.222,Z 350.431,A -85,B 0,C 180,E1 -17971.905,E2 -17971.905} C_VEL
LIN {X 0,Y 269.959,Z 350.465,A -85,B 0,C 180,E1 -17972.737,E2 -17972.737} C_VEL
LIN {X 0,Y 268.633,Z 350.638,A -85,B 0,C 180,E1 -17973.965,E2 -17973.965} C_VEL
LIN {X 0,Y 264.251,Z 351.192,A -85,B 0,C 180,E1 -17976.822,E2 -17976.822} C_VEL
LIN {X 0,Y 263.205,Z 351.312,A -85,B 0,C 180,E1 -17978.102,E2 -17978.102} C_VEL
LIN {X 0,Y 263.133,Z 351.315,A -85,B 0,C 180,E1 -17978.535,E2 -17978.535} C_VEL
LIN {X 0,Y 263.209,Z 351.323,A -85,B 0,C 180,E1 -17982.919,E2 -17982.919} C_VEL
LIN {X 0,Y 263.281,Z 351.296,A -85,B 0,C 180,E1 -17986.098,E2 -17986.098} C_VEL
LIN {X 0,Y 263.465,Z 351.291,A -85,B 0,C 180,E1 -17990.79,E2 -17990.79} C_VEL
LIN {X 0,Y 263.482,Z 351.274,A -85,B 0,C 180,E1 -17993.875,E2 -17993.875} C_VEL
LIN {X 0,Y 263.726,Z 351.255,A -85,B 0,C 180,E1 -17998.472,E2 -17998.472} C_VEL
LIN {X 0,Y 263.72,Z 351.253,A -85,B 0,C 180,E1 -18001.527,E2 -18001.527} C_VEL
LIN {X 0,Y 263.516,Z 351.283,A -85,B 0,C 180,E1 -18007.663,E2 -18007.663} C_VEL
LIN {X 0,Y 263.325,Z 351.299,A -85,B 0,C 180,E1 -18010.767,E2 -18010.767} C_VEL
LIN {X 0,Y 263.315,Z 351.295,A -85,B 0,C 180,E1 -18015.48,E2 -18015.48} C_VEL
LIN {X 0,Y 263.23,Z 351.308,A -85,B 0,C 180,E1 -18020.309,E2 -18020.309} C_VEL
LIN {X 0,Y 263.161,Z 351.321,A -85,B 0,C 180,E1 -18025.296,E2 -18025.296} C_VEL
LIN {X 0,Y 263.127,Z 351.331,A -85,B 0,C 180,E1 -18028.735,E2 -18028.735} C_VEL
LIN {X 0,Y 263.121,Z 351.335,A -85,B 0,C 180,E1 -18032.289,E2 -18032.289} C_VEL
LIN {X 0,Y 263.185,Z 351.324,A -85,B 0,C 180,E1 -18036.766,E2 -18036.766} C_VEL
LIN {X 0,Y 263.119,Z 351.317,A -85,B 0,C 180,E1 -18041.594,E2 -18041.594} C_VEL
LIN {X 0,Y 263.118,Z 351.336,A -85,B 0,C 180,E1 -18046.017,E2 -18046.017} C_VEL
LIN {X 0,Y 263.155,Z 351.373,A -85,B 0,C 180,E1 -18049.638,E2 -18049.638} C_VEL
LIN {X 0,Y 265.808,Z 361.44,A -85,B 0,C 180,E1 -18053.412,E2 -18053.412} C_VEL
LIN {X 0,Y 266.273,Z 363.407,A -85,B 0,C 180,E1 -18054.042,E2 -18054.042} C_VEL
LIN {X 0,Y 275.046,Z 382.508,A -85,B 0,C 180,E1 -18055.804,E2 -18055.804} C_VEL
LIN {X 0,Y 280.601,Z 396.601,A -85,B 0,C 180,E1 -18056.906,E2 -18056.906} C_VEL
LIN {X 0,Y 283.495,Z 417.678,A -85,B 0,C 180,E1 -18057.85,E2 -18057.85} C_VEL
LIN {X 0,Y 280.546,Z 501.163,A -85,B 0,C 180,E1 -18059.933,E2 -18059.933} C_VEL
LIN {X 0,Y 279.442,Z 515.243,A -85,B 0,C 180,E1 -18060.529,E2 -18060.529} C_VEL
LIN {X 0,Y 277.887,Z 528.957,A -85,B 0,C 180,E1 -18061.384,E2 -18061.384} C_VEL
LIN {X 0,Y 275.992,Z 542.279,A -85,B 0,C 180,E1 -18062.514,E2 -18062.514} C_VEL
LIN {X 0,Y 273.92,Z 554.985,A -85,B 0,C 180,E1 -18063.917,E2 -18063.917} C_VEL
LIN {X 0,Y 271.729,Z 566.806,A -85,B 0,C 180,E1 -18065.555,E2 -18065.555} C_VEL
LIN {X 0,Y 269.426,Z 577.493,A -85,B 0,C 180,E1 -18067.372,E2 -18067.372} C_VEL
LIN {X 0,Y 267.162,Z 588.101,A -85,B 0,C 180,E1 -18069.602,E2 -18069.602} C_VEL
LIN {X 0,Y 265.325,Z 596.853,A -85,B 0,C 180,E1 -18071.867,E2 -18071.867} C_VEL
LIN {X 0,Y 263.766,Z 605.239,A -85,B 0,C 180,E1 -18074.547,E2 -18074.547} C_VEL
LIN {X 0,Y 262.627,Z 611.073,A -85,B 0,C 180,E1 -18076.853,E2 -18076.853} C_VEL
LIN {X 0,Y 261.817,Z 615.863,A -85,B 0,C 180,E1 -18079.17,E2 -18079.17} C_VEL
LIN {X 0,Y 261.301,Z 620.82,A -85,B 0,C 180,E1 -18082.272,E2 -18082.272} C_VEL
LIN {X 0,Y 261.073,Z 624.257,A -85,B 0,C 180,E1 -18085.368,E2 -18085.368} C_VEL
LIN {X 0,Y 261.117,Z 626.282,A -85,B 0,C 180,E1 -18088.458,E2 -18088.458} C_VEL
LIN {X 0,Y 261.126,Z 626.78,A -85,B 0,C 180,E1 -18090,E2 -18090} C_VEL
LIN {X 0,Y 261.111,Z 626.939,A -85,B 0,C 180,E1 -18091.542,E2 -18091.542} C_VEL
LIN {X 0,Y 261.045,Z 626.249,A -85,B 0,C 180,E1 -18094.633,E2 -18094.633} C_VEL
LIN {X 0,Y 261.291,Z 624.22,A -85,B 0,C 180,E1 -18097.729,E2 -18097.729} C_VEL
LIN {X 0,Y 261.955,Z 620.808,A -85,B 0,C 180,E1 -18100.824,E2 -18100.824} C_VEL
LIN {X 0,Y 263.23,Z 615.921,A -85,B 0,C 180,E1 -18103.903,E2 -18103.903} C_VEL
LIN {X 0,Y 265.099,Z 609.417,A -85,B 0,C 180,E1 -18106.954,E2 -18106.954} C_VEL
LIN {X 0,Y 267.195,Z 602.203,A -85,B 0,C 180,E1 -18109.594,E2 -18109.594} C_VEL
LIN {X 0,Y 269.957,Z 593.311,A -85,B 0,C 180,E1 -18112.178,E2 -18112.178} C_VEL
LIN {X 0,Y 272.775,Z 584.004,A -85,B 0,C 180,E1 -18114.345,E2 -18114.345} C_VEL
LIN {X 0,Y 275.726,Z 573.725,A -85,B 0,C 180,E1 -18116.287,E2 -18116.287} C_VEL
LIN {X 0,Y 278.629,Z 562.151,A -85,B 0,C 180,E1 -18118.062,E2 -18118.062} C_VEL
LIN {X 0,Y 281.446,Z 549.934,A -85,B 0,C 180,E1 -18119.549,E2 -18119.549} C_VEL
LIN {X 0,Y 283.781,Z 537.877,A -85,B 0,C 180,E1 -18120.716,E2 -18120.716} C_VEL
LIN {X 0,Y 285.983,Z 524.632,A -85,B 0,C 180,E1 -18121.687,E2 -18121.687} C_VEL
LIN {X 0,Y 287.823,Z 510.236,A -85,B 0,C 180,E1 -18122.44,E2 -18122.44} C_VEL
LIN {X 0,Y 288.847,Z 496.308,A -85,B 0,C 180,E1 -18122.928,E2 -18122.928} C_VEL
LIN {X 0,Y 292.029,Z 419.444,A -85,B 0,C 180,E1 -18124.79,E2 -18124.79} C_VEL
LIN {X 0,Y 290.241,Z 408.904,A -85,B 0,C 180,E1 -18125.38,E2 -18125.38} C_VEL
LIN {X 0,Y 283.621,Z 394.205,A -85,B 0,C 180,E1 -18126.893,E2 -18126.893} C_VEL
LIN {X 0,Y 276.679,Z 380.435,A -85,B 0,C 180,E1 -18128.542,E2 -18128.542} C_VEL
LIN {X 0,Y 271.313,Z 370.94,A -85,B 0,C 180,E1 -18129.866,E2 -18129.866} C_VEL
LIN {X 0,Y 268.434,Z 366.105,A -85,B 0,C 180,E1 -18130.601,E2 -18130.601} C_VEL
LIN {X 0,Y 266.449,Z 362.307,A -85,B 0,C 180,E1 -18131.19,E2 -18131.19} C_VEL
LIN {X 0,Y 263.817,Z 353.639,A -85,B 0,C 180,E1 -18135.094,E2 -18135.094} C_VEL
LIN {X 0,Y 263.096,Z 351.335,A -85,B 0,C 180,E1 -18136.279,E2 -18136.279} C_VEL
LIN {X 0,Y 263.1,Z 351.333,A -85,B 0,C 180,E1 -18140.127,E2 -18140.127} C_VEL
LIN {X 0,Y 263.157,Z 351.33,A -85,B 0,C 180,E1 -18144.018,E2 -18144.018} C_VEL
LIN {X 0,Y 263.12,Z 351.326,A -85,B 0,C 180,E1 -18147.71,E2 -18147.71} C_VEL
LIN {X 0,Y 263.135,Z 351.311,A -85,B 0,C 180,E1 -18151.807,E2 -18151.807} C_VEL
LIN {X 0,Y 263.182,Z 351.317,A -85,B 0,C 180,E1 -18155.218,E2 -18155.218} C_VEL
LIN {X 0,Y 263.231,Z 351.311,A -85,B 0,C 180,E1 -18159.691,E2 -18159.691} C_VEL
LIN {X 0,Y 263.315,Z 351.302,A -85,B 0,C 180,E1 -18164.52,E2 -18164.52} C_VEL
LIN {X 0,Y 263.325,Z 351.3,A -85,B 0,C 180,E1 -18169.233,E2 -18169.233} C_VEL
LIN {X 0,Y 263.517,Z 351.275,A -85,B 0,C 180,E1 -18172.337,E2 -18172.337} C_VEL
LIN {X 0,Y 263.73,Z 351.247,A -85,B 0,C 180,E1 -18178.473,E2 -18178.473} C_VEL
LIN {X 0,Y 263.727,Z 351.252,A -85,B 0,C 180,E1 -18181.528,E2 -18181.528} C_VEL
LIN {X 0,Y 263.525,Z 351.272,A -85,B 0,C 180,E1 -18187.664,E2 -18187.664} C_VEL
LIN {X 0,Y 263.339,Z 351.303,A -85,B 0,C 180,E1 -18190.768,E2 -18190.768} C_VEL
LIN {X 0,Y 263.304,Z 351.306,A -85,B 0,C 180,E1 -18195.481,E2 -18195.481} C_VEL
LIN {X 0,Y 263.204,Z 351.315,A -85,B 0,C 180,E1 -18200.312,E2 -18200.312} C_VEL
LIN {X 0,Y 263.188,Z 351.321,A -85,B 0,C 180,E1 -18205.294,E2 -18205.294} C_VEL
LIN {X 0,Y 263.171,Z 351.322,A -85,B 0,C 180,E1 -18208.731,E2 -18208.731} C_VEL
LIN {X 0,Y 263.129,Z 351.329,A -85,B 0,C 180,E1 -18212.29,E2 -18212.29} C_VEL
LIN {X 0,Y 263.18,Z 351.321,A -85,B 0,C 180,E1 -18216.764,E2 -18216.764} C_VEL
LIN {X 0,Y 263.122,Z 351.334,A -85,B 0,C 180,E1 -18221.595,E2 -18221.595} C_VEL
LIN {X 0,Y 263.141,Z 351.465,A -85,B 0,C 180,E1 -18222.02,E2 -18222.02} C_VEL
LIN {X 0,Y 263.269,Z 352.074,A -85,B 0,C 180,E1 -18222.252,E2 -18222.252} C_VEL
LIN {X 0,Y 264.447,Z 354.655,A -85,B 0,C 180,E1 -18222.6,E2 -18222.6} C_VEL
LIN {X 0,Y 266.456,Z 357.152,A -85,B 0,C 180,E1 -18223.111,E2 -18223.111} C_VEL
LIN {X 0,Y 272.525,Z 366.67,A -85,B 0,C 180,E1 -18224.654,E2 -18224.654} C_VEL
LIN {X 0,Y 279.648,Z 379.02,A -85,B 0,C 180,E1 -18226.374,E2 -18226.374} C_VEL
LIN {X 0,Y 286.372,Z 391.75,A -85,B 0,C 180,E1 -18227.915,E2 -18227.915} C_VEL
LIN {X 0,Y 292.576,Z 405.441,A -85,B 0,C 180,E1 -18229.305,E2 -18229.305} C_VEL
LIN {X 0,Y 289.05,Z 487.83,A -85,B 0,C 180,E1 -18231.317,E2 -18231.317} C_VEL
LIN {X 0,Y 287.769,Z 502.516,A -85,B 0,C 180,E1 -18231.946,E2 -18231.946} C_VEL
LIN {X 0,Y 285.925,Z 516.98,A -85,B 0,C 180,E1 -18232.863,E2 -18232.863} C_VEL
LIN {X 0,Y 283.764,Z 529.948,A -85,B 0,C 180,E1 -18233.971,E2 -18233.971} C_VEL
LIN {X 0,Y 281.225,Z 542.287,A -85,B 0,C 180,E1 -18235.319,E2 -18235.319} C_VEL
LIN {X 0,Y 278.371,Z 553.95,A -85,B 0,C 180,E1 -18236.91,E2 -18236.91} C_VEL
LIN {X 0,Y 275.794,Z 563.454,A -85,B 0,C 180,E1 -18238.508,E2 -18238.508} C_VEL
LIN {X 0,Y 272.832,Z 574.031,A -85,B 0,C 180,E1 -18240.698,E2 -18240.698} C_VEL
LIN {X 0,Y 270.328,Z 582.726,A -85,B 0,C 180,E1 -18242.938,E2 -18242.938} C_VEL
LIN {X 0,Y 267.585,Z 591.012,A -85,B 0,C 180,E1 -18245.565,E2 -18245.565} C_VEL
LIN {X 0,Y 265.457,Z 597.635,A -85,B 0,C 180,E1 -18248.245,E2 -18248.245} C_VEL
LIN {X 0,Y 263.596,Z 603.484,A -85,B 0,C 180,E1 -18251.341,E2 -18251.341} C_VEL
LIN {X 0,Y 262.334,Z 607.734,A -85,B 0,C 180,E1 -18254.461,E2 -18254.461} C_VEL
LIN {X 0,Y 261.442,Z 610.52,A -85,B 0,C 180,E1 -18257.582,E2 -18257.582} C_VEL
LIN {X 0,Y 261.085,Z 611.928,A -85,B 0,C 180,E1 -18260.706,E2 -18260.706} C_VEL
LIN {X 0,Y 261.091,Z 612.002,A -85,B 0,C 180,E1 -18263.819,E2 -18263.819} C_VEL
LIN {X 0,Y 261.147,Z 610.759,A -85,B 0,C 180,E1 -18266.915,E2 -18266.915} C_VEL
LIN {X 0,Y 261.287,Z 608.174,A -85,B 0,C 180,E1 -18270,E2 -18270} C_VEL
LIN {X 0,Y 261.79,Z 604.171,A -85,B 0,C 180,E1 -18273.078,E2 -18273.078} C_VEL
LIN {X 0,Y 262.599,Z 600.186,A -85,B 0,C 180,E1 -18275.375,E2 -18275.375} C_VEL
LIN {X 0,Y 263.467,Z 595.237,A -85,B 0,C 180,E1 -18277.664,E2 -18277.664} C_VEL
LIN {X 0,Y 265.138,Z 588.144,A -85,B 0,C 180,E1 -18280.307,E2 -18280.307} C_VEL
LIN {X 0,Y 266.866,Z 580.558,A -85,B 0,C 180,E1 -18282.598,E2 -18282.598} C_VEL
LIN {X 0,Y 268.652,Z 571.85,A -85,B 0,C 180,E1 -18284.777,E2 -18284.777} C_VEL
LIN {X 0,Y 270.526,Z 563.024,A -85,B 0,C 180,E1 -18286.604,E2 -18286.604} C_VEL
LIN {X 0,Y 272.919,Z 551.334,A -85,B 0,C 180,E1 -18288.582,E2 -18288.582} C_VEL
LIN {X 0,Y 275,Z 539.62,A -85,B 0,C 180,E1 -18290.182,E2 -18290.182} C_VEL
LIN {X 0,Y 277.061,Z 526.695,A -85,B 0,C 180,E1 -18291.58,E2 -18291.58} C_VEL
LIN {X 0,Y 278.788,Z 513.169,A -85,B 0,C 180,E1 -18292.706,E2 -18292.706} C_VEL
LIN {X 0,Y 280.128,Z 499.783,A -85,B 0,C 180,E1 -18293.519,E2 -18293.519} C_VEL
LIN {X 0,Y 280.997,Z 486.413,A -85,B 0,C 180,E1 -18294.078,E2 -18294.078} C_VEL
LIN {X 0,Y 283.984,Z 396.855,A -85,B 0,C 180,E1 -18296.325,E2 -18296.325} C_VEL
LIN {X 0,Y 276.081,Z 377.505,A -85,B 0,C 180,E1 -18297.851,E2 -18297.851} C_VEL
LIN {X 0,Y 268.598,Z 361.696,A -85,B 0,C 180,E1 -18299.325,E2 -18299.325} C_VEL
LIN {X 0,Y 264.697,Z 354.848,A -85,B 0,C 180,E1 -18300.092,E2 -18300.092} C_VEL
LIN {X 0,Y 263.428,Z 352.388,A -85,B 0,C 180,E1 -18300.355,E2 -18300.355} C_VEL
LIN {X 0,Y 263.197,Z 351.326,A -85,B 0,C 180,E1 -18300.453,E2 -18300.453} C_VEL
LIN {X 0,Y 263.174,Z 351.327,A -85,B 0,C 180,E1 -18304.12,E2 -18304.12} C_VEL
LIN {X 0,Y 263.166,Z 351.33,A -85,B 0,C 180,E1 -18307.895,E2 -18307.895} C_VEL
LIN {X 0,Y 263.123,Z 351.323,A -85,B 0,C 180,E1 -18311.892,E2 -18311.892} C_VEL
LIN {X 0,Y 263.103,Z 351.337,A -85,B 0,C 180,E1 -18316.154,E2 -18316.154} C_VEL
LIN {X 0,Y 263.103,Z 351.337,A -85,B 0,C 180,E1 -18320.126,E2 -18320.126} C_VEL
LIN {X 0,Y 263.159,Z 351.329,A -85,B 0,C 180,E1 -18324.017,E2 -18324.017} C_VEL
LIN {X 0,Y 263.129,Z 351.328,A -85,B 0,C 180,E1 -18327.71,E2 -18327.71} C_VEL
LIN {X 0,Y 263.17,Z 351.31,A -85,B 0,C 180,E1 -18331.893,E2 -18331.893} C_VEL
LIN {X 0,Y 263.193,Z 351.324,A -85,B 0,C 180,E1 -18335.213,E2 -18335.213} C_VEL
LIN {X 0,Y 263.133,Z 351.315,A -85,B 0,C 180,E1 -18338.535,E2 -18338.535} C_VEL
LIN {X 0,Y 262.502,Z 351.391,A -85,B 0,C 180,E1 -18339.813,E2 -18339.813} C_VEL
LIN {X 0,Y 259.677,Z 351.758,A -85,B 0,C 180,E1 -18341.897,E2 -18341.897} C_VEL
LIN {X 0,Y 257.277,Z 352.061,A -85,B 0,C 180,E1 -18343.592,E2 -18343.592} C_VEL
LIN {X 0,Y 256.273,Z 352.18,A -85,B 0,C 180,E1 -18344.906,E2 -18344.906} C_VEL
LIN {X 0,Y 256.206,Z 352.183,A -85,B 0,C 180,E1 -18345.351,E2 -18345.351} C_VEL
LIN {X 0,Y 256.28,Z 352.169,A -85,B 0,C 180,E1 -18348.932,E2 -18348.932} C_VEL
LIN {X 0,Y 256.49,Z 352.16,A -85,B 0,C 180,E1 -18352.125,E2 -18352.125} C_VEL
LIN {X 0,Y 256.447,Z 352.145,A -85,B 0,C 180,E1 -18356.857,E2 -18356.857} C_VEL
LIN {X 0,Y 256.688,Z 352.131,A -85,B 0,C 180,E1 -18358.431,E2 -18358.431} C_VEL
LIN {X 0,Y 256.681,Z 352.129,A -85,B 0,C 180,E1 -18361.568,E2 -18361.568} C_VEL
LIN {X 0,Y 256.443,Z 352.168,A -85,B 0,C 180,E1 -18366.293,E2 -18366.293} C_VEL
LIN {X 0,Y 256.394,Z 352.155,A -85,B 0,C 180,E1 -18369.466,E2 -18369.466} C_VEL
LIN {X 0,Y 256.228,Z 352.185,A -85,B 0,C 180,E1 -18374.291,E2 -18374.291} C_VEL
LIN {X 0,Y 256.17,Z 352.196,A -85,B 0,C 180,E1 -18377.564,E2 -18377.564} C_VEL
LIN {X 0,Y 256.133,Z 352.188,A -85,B 0,C 180,E1 -18381.11,E2 -18381.11} C_VEL
LIN {X 0,Y 256.126,Z 352.199,A -85,B 0,C 180,E1 -18385.112,E2 -18385.112} C_VEL
LIN {X 0,Y 256.048,Z 352.21,A -85,B 0,C 180,E1 -18389.608,E2 -18389.608} C_VEL
LIN {X 0,Y 256.06,Z 352.212,A -85,B 0,C 180,E1 -18393.293,E2 -18393.293} C_VEL
LIN {X 0,Y 256.115,Z 352.203,A -85,B 0,C 180,E1 -18397.273,E2 -18397.273} C_VEL
LIN {X 0,Y 256.066,Z 352.197,A -85,B 0,C 180,E1 -18402.182,E2 -18402.182} C_VEL
LIN {X 0,Y 256.057,Z 352.213,A -85,B 0,C 180,E1 -18406.674,E2 -18406.674} C_VEL
LIN {X 0,Y 256.114,Z 352.252,A -85,B 0,C 180,E1 -18408.81,E2 -18408.81} C_VEL
LIN {X 0,Y 258.908,Z 362.921,A -85,B 0,C 180,E1 -18412.954,E2 -18412.954} C_VEL
LIN {X 0,Y 268.132,Z 382.679,A -85,B 0,C 180,E1 -18414.902,E2 -18414.902} C_VEL
LIN {X 0,Y 274.604,Z 398.589,A -85,B 0,C 180,E1 -18416.23,E2 -18416.23} C_VEL
LIN {X 0,Y 277.301,Z 418.824,A -85,B 0,C 180,E1 -18417.16,E2 -18417.16} C_VEL
LIN {X 0,Y 274.243,Z 501.646,A -85,B 0,C 180,E1 -18419.275,E2 -18419.275} C_VEL
LIN {X 0,Y 273.092,Z 515.479,A -85,B 0,C 180,E1 -18419.88,E2 -18419.88} C_VEL
LIN {X 0,Y 271.482,Z 529.081,A -85,B 0,C 180,E1 -18420.751,E2 -18420.751} C_VEL
LIN {X 0,Y 269.692,Z 541.446,A -85,B 0,C 180,E1 -18421.816,E2 -18421.816} C_VEL
LIN {X 0,Y 267.679,Z 553.523,A -85,B 0,C 180,E1 -18423.151,E2 -18423.151} C_VEL
LIN {X 0,Y 265.185,Z 566.18,A -85,B 0,C 180,E1 -18424.911,E2 -18424.911} C_VEL
LIN {X 0,Y 262.849,Z 576.945,A -85,B 0,C 180,E1 -18426.773,E2 -18426.773} C_VEL
LIN {X 0,Y 260.469,Z 587.611,A -85,B 0,C 180,E1 -18429.053,E2 -18429.053} C_VEL
LIN {X 0,Y 258.522,Z 596.408,A -85,B 0,C 180,E1 -18431.372,E2 -18431.372} C_VEL
LIN {X 0,Y 256.888,Z 604.849,A -85,B 0,C 180,E1 -18434.123,E2 -18434.123} C_VEL
LIN {X 0,Y 255.682,Z 610.711,A -85,B 0,C 180,E1 -18436.489,E2 -18436.489} C_VEL
LIN {X 0,Y 254.795,Z 615.534,A -85,B 0,C 180,E1 -18438.868,E2 -18438.868} C_VEL
LIN {X 0,Y 254.234,Z 620.524,A -85,B 0,C 180,E1 -18442.055,E2 -18442.055} C_VEL
LIN {X 0,Y 254.012,Z 623.992,A -85,B 0,C 180,E1 -18445.239,E2 -18445.239} C_VEL
LIN {X 0,Y 254.023,Z 626.046,A -85,B 0,C 180,E1 -18448.415,E2 -18448.415} C_VEL
LIN {X 0,Y 254.054,Z 626.56,A -85,B 0,C 180,E1 -18450,E2 -18450} C_VEL
LIN {X 0,Y 254.016,Z 626.735,A -85,B 0,C 180,E1 -18451.585,E2 -18451.585} C_VEL
LIN {X 0,Y 253.952,Z 626.078,A -85,B 0,C 180,E1 -18454.762,E2 -18454.762} C_VEL
LIN {X 0,Y 254.23,Z 624.081,A -85,B 0,C 180,E1 -18457.945,E2 -18457.945} C_VEL
LIN {X 0,Y 254.949,Z 620.699,A -85,B 0,C 180,E1 -18461.126,E2 -18461.126} C_VEL
LIN {X 0,Y 256.303,Z 615.843,A -85,B 0,C 180,E1 -18464.287,E2 -18464.287} C_VEL
LIN {X 0,Y 258.251,Z 609.375,A -85,B 0,C 180,E1 -18467.418,E2 -18467.418} C_VEL
LIN {X 0,Y 260.48,Z 602.2,A -85,B 0,C 180,E1 -18470.121,E2 -18470.121} C_VEL
LIN {X 0,Y 262.941,Z 594.707,A -85,B 0,C 180,E1 -18472.388,E2 -18472.388} C_VEL
LIN {X 0,Y 265.795,Z 585.731,A -85,B 0,C 180,E1 -18474.61,E2 -18474.61} C_VEL
LIN {X 0,Y 269.088,Z 574.88,A -85,B 0,C 180,E1 -18476.777,E2 -18476.777} C_VEL
LIN {X 0,Y 271.986,Z 564.02,A -85,B 0,C 180,E1 -18478.533,E2 -18478.533} C_VEL
LIN {X 0,Y 274.98,Z 551.85,A -85,B 0,C 180,E1 -18480.104,E2 -18480.104} C_VEL
LIN {X 0,Y 277.348,Z 540.282,A -85,B 0,C 180,E1 -18481.296,E2 -18481.296} C_VEL
LIN {X 0,Y 279.823,Z 526.651,A -85,B 0,C 180,E1 -18482.362,E2 -18482.362} C_VEL
LIN {X 0,Y 281.795,Z 512.251,A -85,B 0,C 180,E1 -18483.169,E2 -18483.169} C_VEL
LIN {X 0,Y 283.027,Z 498.181,A -85,B 0,C 180,E1 -18483.696,E2 -18483.696} C_VEL
LIN {X 0,Y 286.369,Z 420.62,A -85,B 0,C 180,E1 -18485.616,E2 -18485.616} C_VEL
LIN {X 0,Y 284.925,Z 411.898,A -85,B 0,C 180,E1 -18486.118,E2 -18486.118} C_VEL
LIN {X 0,Y 278.225,Z 396.925,A -85,B 0,C 180,E1 -18487.719,E2 -18487.719} C_VEL
LIN {X 0,Y 270.233,Z 381.16,A -85,B 0,C 180,E1 -18489.714,E2 -18489.714} C_VEL
LIN {X 0,Y 261.861,Z 366.792,A -85,B 0,C 180,E1 -18491.933,E2 -18491.933} C_VEL
LIN {X 0,Y 259.241,Z 362.549,A -85,B 0,C 180,E1 -18492.666,E2 -18492.666} C_VEL
LIN {X 0,Y 258.977,Z 361.801,A -85,B 0,C 180,E1 -18492.886,E2 -18492.886} C_VEL
LIN {X 0,Y 257.006,Z 355.406,A -85,B 0,C 180,E1 -18495.927,E2 -18495.927} C_VEL
LIN {X 0,Y 256.086,Z 352.204,A -85,B 0,C 180,E1 -18497.634,E2 -18497.634} C_VEL
LIN {X 0,Y 256.066,Z 352.214,A -85,B 0,C 180,E1 -18500.857,E2 -18500.857} C_VEL
LIN {X 0,Y 256.125,Z 352.202,A -85,B 0,C 180,E1 -18502.867,E2 -18502.867} C_VEL
LIN {X 0,Y 256.059,Z 352.214,A -85,B 0,C 180,E1 -18506.706,E2 -18506.706} C_VEL
LIN {X 0,Y 256.036,Z 352.18,A -85,B 0,C 180,E1 -18510.391,E2 -18510.391} C_VEL
LIN {X 0,Y 256.126,Z 352.197,A -85,B 0,C 180,E1 -18514.888,E2 -18514.888} C_VEL
LIN {X 0,Y 256.14,Z 352.194,A -85,B 0,C 180,E1 -18519.103,E2 -18519.103} C_VEL
LIN {X 0,Y 256.238,Z 352.181,A -85,B 0,C 180,E1 -18524.082,E2 -18524.082} C_VEL
LIN {X 0,Y 256.271,Z 352.176,A -85,B 0,C 180,E1 -18528.933,E2 -18528.933} C_VEL
LIN {X 0,Y 256.46,Z 352.155,A -85,B 0,C 180,E1 -18532.125,E2 -18532.125} C_VEL
LIN {X 0,Y 256.442,Z 352.158,A -85,B 0,C 180,E1 -18536.858,E2 -18536.858} C_VEL
LIN {X 0,Y 256.692,Z 352.123,A -85,B 0,C 180,E1 -18538.432,E2 -18538.432} C_VEL
LIN {X 0,Y 256.69,Z 352.128,A -85,B 0,C 180,E1 -18541.569,E2 -18541.569} C_VEL
LIN {X 0,Y 256.444,Z 352.157,A -85,B 0,C 180,E1 -18546.695,E2 -18546.695} C_VEL
LIN {X 0,Y 256.396,Z 352.173,A -85,B 0,C 180,E1 -18549.467,E2 -18549.467} C_VEL
LIN {X 0,Y 256.225,Z 352.194,A -85,B 0,C 180,E1 -18554.292,E2 -18554.292} C_VEL
LIN {X 0,Y 256.157,Z 352.196,A -85,B 0,C 180,E1 -18557.566,E2 -18557.566} C_VEL
LIN {X 0,Y 256.118,Z 352.198,A -85,B 0,C 180,E1 -18561.101,E2 -18561.101} C_VEL
LIN {X 0,Y 256.166,Z 352.194,A -85,B 0,C 180,E1 -18565.131,E2 -18565.131} C_VEL
LIN {X 0,Y 256.107,Z 352.209,A -85,B 0,C 180,E1 -18569.601,E2 -18569.601} C_VEL
LIN {X 0,Y 256.064,Z 352.212,A -85,B 0,C 180,E1 -18573.294,E2 -18573.294} C_VEL
LIN {X 0,Y 256.112,Z 352.2,A -85,B 0,C 180,E1 -18577.272,E2 -18577.272} C_VEL
LIN {X 0,Y 256.054,Z 352.21,A -85,B 0,C 180,E1 -18580.619,E2 -18580.619} C_VEL
LIN {X 0,Y 257.007,Z 354.965,A -85,B 0,C 180,E1 -18580.97,E2 -18580.97} C_VEL
LIN {X 0,Y 259.35,Z 357.67,A -85,B 0,C 180,E1 -18581.607,E2 -18581.607} C_VEL
LIN {X 0,Y 261.518,Z 360.99,A -85,B 0,C 180,E1 -18582.211,E2 -18582.211} C_VEL
LIN {X 0,Y 263.067,Z 363.279,A -85,B 0,C 180,E1 -18582.629,E2 -18582.629} C_VEL
LIN {X 0,Y 268.618,Z 372.031,A -85,B 0,C 180,E1 -18584.085,E2 -18584.085} C_VEL
LIN {X 0,Y 275.573,Z 384.272,A -85,B 0,C 180,E1 -18585.825,E2 -18585.825} C_VEL
LIN {X 0,Y 283.146,Z 399.092,A -85,B 0,C 180,E1 -18587.622,E2 -18587.622} C_VEL
LIN {X 0,Y 286.928,Z 407.687,A -85,B 0,C 180,E1 -18588.505,E2 -18588.505} C_VEL
LIN {X 0,Y 283.271,Z 488.384,A -85,B 0,C 180,E1 -18590.503,E2 -18590.503} C_VEL
LIN {X 0,Y 281.943,Z 503,A -85,B 0,C 180,E1 -18591.144,E2 -18591.144} C_VEL
LIN {X 0,Y 280.056,Z 517.229,A -85,B 0,C 180,E1 -18592.062,E2 -18592.062} C_VEL
LIN {X 0,Y 277.97,Z 529.291,A -85,B 0,C 180,E1 -18593.097,E2 -18593.097} C_VEL
LIN {X 0,Y 275.25,Z 542.103,A -85,B 0,C 180,E1 -18594.502,E2 -18594.502} C_VEL
LIN {X 0,Y 272.366,Z 553.583,A -85,B 0,C 180,E1 -18596.083,E2 -18596.083} C_VEL
LIN {X 0,Y 270.185,Z 561.211,A -85,B 0,C 180,E1 -18597.335,E2 -18597.335} C_VEL
LIN {X 0,Y 267.001,Z 572.196,A -85,B 0,C 180,E1 -18599.557,E2 -18599.557} C_VEL
LIN {X 0,Y 264.317,Z 581.236,A -85,B 0,C 180,E1 -18601.839,E2 -18601.839} C_VEL
LIN {X 0,Y 261.388,Z 589.849,A -85,B 0,C 180,E1 -18604.521,E2 -18604.521} C_VEL
LIN {X 0,Y 259.039,Z 596.835,A -85,B 0,C 180,E1 -18607.29,E2 -18607.29} C_VEL
LIN {X 0,Y 257.216,Z 602.225,A -85,B 0,C 180,E1 -18610.03,E2 -18610.03} C_VEL
LIN {X 0,Y 255.995,Z 605.873,A -85,B 0,C 180,E1 -18612.423,E2 -18612.423} C_VEL
LIN {X 0,Y 254.858,Z 609.417,A -85,B 0,C 180,E1 -18615.63,E2 -18615.63} C_VEL
LIN {X 0,Y 254.11,Z 611.548,A -85,B 0,C 180,E1 -18618.837,E2 -18618.837} C_VEL
LIN {X 0,Y 253.955,Z 612.324,A -85,B 0,C 180,E1 -18622.047,E2 -18622.047} C_VEL
LIN {X 0,Y 254.017,Z 611.777,A -85,B 0,C 180,E1 -18625.239,E2 -18625.239} C_VEL
LIN {X 0,Y 254.121,Z 609.916,A -85,B 0,C 180,E1 -18628.415,E2 -18628.415} C_VEL
LIN {X 0,Y 254.425,Z 606.684,A -85,B 0,C 180,E1 -18631.583,E2 -18631.583} C_VEL
LIN {X 0,Y 255.164,Z 601.978,A -85,B 0,C 180,E1 -18634.74,E2 -18634.74} C_VEL
LIN {X 0,Y 256.46,Z 595.657,A -85,B 0,C 180,E1 -18637.875,E2 -18637.875} C_VEL
LIN {X 0,Y 258.18,Z 588.615,A -85,B 0,C 180,E1 -18640.588,E2 -18640.588} C_VEL
LIN {X 0,Y 260.242,Z 579.929,A -85,B 0,C 180,E1 -18643.267,E2 -18643.267} C_VEL
LIN {X 0,Y 262.195,Z 570.83,A -85,B 0,C 180,E1 -18645.547,E2 -18645.547} C_VEL
LIN {X 0,Y 264.207,Z 561.757,A -85,B 0,C 180,E1 -18647.412,E2 -18647.412} C_VEL
LIN {X 0,Y 266.496,Z 550.931,A -85,B 0,C 180,E1 -18649.247,E2 -18649.247} C_VEL
LIN {X 0,Y 268.636,Z 539.09,A -85,B 0,C 180,E1 -18650.882,E2 -18650.882} C_VEL
LIN {X 0,Y 270.807,Z 525.959,A -85,B 0,C 180,E1 -18652.305,E2 -18652.305} C_VEL
LIN {X 0,Y 272.46,Z 513.318,A -85,B 0,C 180,E1 -18653.365,E2 -18653.365} C_VEL
LIN {X 0,Y 273.834,Z 499.91,A -85,B 0,C 180,E1 -18654.194,E2 -18654.194} C_VEL
LIN {X 0,Y 274.746,Z 486.489,A -85,B 0,C 180,E1 -18654.763,E2 -18654.763} C_VEL
LIN {X 0,Y 277.784,Z 398.661,A -85,B 0,C 180,E1 -18657.011,E2 -18657.011} C_VEL
LIN {X 0,Y 270.46,Z 380.707,A -85,B 0,C 180,E1 -18658.484,E2 -18658.484} C_VEL
LIN {X 0,Y 263.613,Z 366.038,A -85,B 0,C 180,E1 -18659.89,E2 -18659.89} C_VEL
LIN {X 0,Y 259.144,Z 358.264,A -85,B 0,C 180,E1 -18660.801,E2 -18660.801} C_VEL
LIN {X 0,Y 257.574,Z 355.73,A -85,B 0,C 180,E1 -18661.124,E2 -18661.124} C_VEL
LIN {X 0,Y 256.296,Z 353.21,A -85,B 0,C 180,E1 -18661.406,E2 -18661.406} C_VEL
LIN {X 0,Y 256.094,Z 352.21,A -85,B 0,C 180,E1 -18661.494,E2 -18661.494} C_VEL
LIN {X 0,Y 256.121,Z 352.195,A -85,B 0,C 180,E1 -18665.186,E2 -18665.186} C_VEL
LIN {X 0,Y 256.087,Z 352.197,A -85,B 0,C 180,E1 -18669.138,E2 -18669.138} C_VEL
LIN {X 0,Y 256.048,Z 352.217,A -85,B 0,C 180,E1 -18673.328,E2 -18673.328} C_VEL
LIN {X 0,Y 256.068,Z 352.206,A -85,B 0,C 180,E1 -18677.818,E2 -18677.818} C_VEL
LIN {X 0,Y 256.069,Z 352.213,A -85,B 0,C 180,E1 -18680.857,E2 -18680.857} C_VEL
LIN {X 0,Y 256.126,Z 352.197,A -85,B 0,C 180,E1 -18682.866,E2 -18682.866} C_VEL
LIN {X 0,Y 256.064,Z 352.204,A -85,B 0,C 180,E1 -18686.706,E2 -18686.706} C_VEL
LIN {X 0,Y 256.094,Z 352.207,A -85,B 0,C 180,E1 -18690.397,E2 -18690.397} C_VEL
LIN {X 0,Y 256.162,Z 352.197,A -85,B 0,C 180,E1 -18694.871,E2 -18694.871} C_VEL
LIN {X 0,Y 256.118,Z 352.184,A -85,B 0,C 180,E1 -18699.1,E2 -18699.1} C_VEL
LIN {X 0,Y 256.224,Z 352.192,A -85,B 0,C 180,E1 -18704.08,E2 -18704.08} C_VEL
LIN {X 0,Y 256.206,Z 352.183,A -85,B 0,C 180,E1 -18705.351,E2 -18705.351} C_VEL
LIN {X 0,Y 255.605,Z 352.258,A -85,B 0,C 180,E1 -18706.664,E2 -18706.664} C_VEL
LIN {X 0,Y 252.876,Z 352.608,A -85,B 0,C 180,E1 -18708.807,E2 -18708.807} C_VEL
LIN {X 0,Y 250.524,Z 352.905,A -85,B 0,C 180,E1 -18710.55,E2 -18710.55} C_VEL
LIN {X 0,Y 249.5,Z 353.03,A -85,B 0,C 180,E1 -18711.899,E2 -18711.899} C_VEL
LIN {X 0,Y 249.409,Z 353.036,A -85,B 0,C 180,E1 -18712.356,E2 -18712.356} C_VEL
LIN {X 0,Y 249.65,Z 353.007,A -85,B 0,C 180,E1 -18718.386,E2 -18718.386} C_VEL
LIN {X 0,Y 249.641,Z 353.005,A -85,B 0,C 180,E1 -18721.613,E2 -18721.613} C_VEL
LIN {X 0,Y 249.415,Z 353.043,A -85,B 0,C 180,E1 -18726.471,E2 -18726.471} C_VEL
LIN {X 0,Y 249.326,Z 353.035,A -85,B 0,C 180,E1 -18729.737,E2 -18729.737} C_VEL
LIN {X 0,Y 249.17,Z 353.06,A -85,B 0,C 180,E1 -18734.705,E2 -18734.705} C_VEL
LIN {X 0,Y 249.104,Z 353.079,A -85,B 0,C 180,E1 -18738.079,E2 -18738.079} C_VEL
LIN {X 0,Y 249.073,Z 353.068,A -85,B 0,C 180,E1 -18741.519,E2 -18741.519} C_VEL
LIN {X 0,Y 249.078,Z 353.073,A -85,B 0,C 180,E1 -18745.46,E2 -18745.46} C_VEL
LIN {X 0,Y 249.03,Z 353.087,A -85,B 0,C 180,E1 -18748.974,E2 -18748.974} C_VEL
LIN {X 0,Y 249.021,Z 353.091,A -85,B 0,C 180,E1 -18752.427,E2 -18752.427} C_VEL
LIN {X 0,Y 249.048,Z 353.086,A -85,B 0,C 180,E1 -18756.342,E2 -18756.342} C_VEL
LIN {X 0,Y 249.001,Z 353.08,A -85,B 0,C 180,E1 -18760.479,E2 -18760.479} C_VEL
LIN {X 0,Y 248.998,Z 353.091,A -85,B 0,C 180,E1 -18764.88,E2 -18764.88} C_VEL
LIN {X 0,Y 249.049,Z 353.24,A -85,B 0,C 180,E1 -18767.962,E2 -18767.962} C_VEL
LIN {X 0,Y 251.632,Z 362.821,A -85,B 0,C 180,E1 -18771.816,E2 -18771.816} C_VEL
LIN {X 0,Y 259.869,Z 379.814,A -85,B 0,C 180,E1 -18773.649,E2 -18773.649} C_VEL
LIN {X 0,Y 267.61,Z 398.108,A -85,B 0,C 180,E1 -18775.311,E2 -18775.311} C_VEL
LIN {X 0,Y 268.852,Z 401.633,A -85,B 0,C 180,E1 -18775.584,E2 -18775.584} C_VEL
LIN {X 0,Y 271.18,Z 419.469,A -85,B 0,C 180,E1 -18776.428,E2 -18776.428} C_VEL
LIN {X 0,Y 268.044,Z 500.925,A -85,B 0,C 180,E1 -18778.539,E2 -18778.539} C_VEL
LIN {X 0,Y 266.87,Z 514.943,A -85,B 0,C 180,E1 -18779.157,E2 -18779.157} C_VEL
LIN {X 0,Y 265.122,Z 529.2,A -85,B 0,C 180,E1 -18780.088,E2 -18780.088} C_VEL
LIN {X 0,Y 263.109,Z 542.383,A -85,B 0,C 180,E1 -18781.263,E2 -18781.263} C_VEL
LIN {X 0,Y 260.697,Z 555.807,A -85,B 0,C 180,E1 -18782.826,E2 -18782.826} C_VEL
LIN {X 0,Y 258.256,Z 567.925,A -85,B 0,C 180,E1 -18784.621,E2 -18784.621} C_VEL
LIN {X 0,Y 255.816,Z 578.357,A -85,B 0,C 180,E1 -18786.525,E2 -18786.525} C_VEL
LIN {X 0,Y 253.414,Z 588.737,A -85,B 0,C 180,E1 -18788.868,E2 -18788.868} C_VEL
LIN {X 0,Y 251.434,Z 597.311,A -85,B 0,C 180,E1 -18791.25,E2 -18791.25} C_VEL
LIN {X 0,Y 249.754,Z 605.497,A -85,B 0,C 180,E1 -18794.077,E2 -18794.077} C_VEL
LIN {X 0,Y 248.338,Z 612.079,A -85,B 0,C 180,E1 -18796.915,E2 -18796.915} C_VEL
LIN {X 0,Y 247.396,Z 617.914,A -85,B 0,C 180,E1 -18800.186,E2 -18800.186} C_VEL
LIN {X 0,Y 246.972,Z 622.158,A -85,B 0,C 180,E1 -18803.464,E2 -18803.464} C_VEL
LIN {X 0,Y 246.884,Z 624.939,A -85,B 0,C 180,E1 -18806.736,E2 -18806.736} C_VEL
LIN {X 0,Y 246.983,Z 626.338,A -85,B 0,C 180,E1 -18810,E2 -18810} C_VEL
LIN {X 0,Y 246.848,Z 626.381,A -85,B 0,C 180,E1 -18813.264,E2 -18813.264} C_VEL
LIN {X 0,Y 246.97,Z 625.091,A -85,B 0,C 180,E1 -18816.536,E2 -18816.536} C_VEL
LIN {X 0,Y 247.511,Z 622.444,A -85,B 0,C 180,E1 -18819.809,E2 -18819.809} C_VEL
LIN {X 0,Y 248.509,Z 618.371,A -85,B 0,C 180,E1 -18823.076,E2 -18823.076} C_VEL
LIN {X 0,Y 250.328,Z 612.764,A -85,B 0,C 180,E1 -18826.305,E2 -18826.305} C_VEL
LIN {X 0,Y 252.048,Z 607.391,A -85,B 0,C 180,E1 -18828.736,E2 -18828.736} C_VEL
LIN {X 0,Y 254.637,Z 599.871,A -85,B 0,C 180,E1 -18831.45,E2 -18831.45} C_VEL
LIN {X 0,Y 257.311,Z 591.973,A -85,B 0,C 180,E1 -18833.757,E2 -18833.757} C_VEL
LIN {X 0,Y 260.452,Z 582.467,A -85,B 0,C 180,E1 -18836.007,E2 -18836.007} C_VEL
LIN {X 0,Y 263.694,Z 571.955,A -85,B 0,C 180,E1 -18838.017,E2 -18838.017} C_VEL
LIN {X 0,Y 266.86,Z 560.148,A -85,B 0,C 180,E1 -18839.844,E2 -18839.844} C_VEL
LIN {X 0,Y 269.866,Z 547.517,A -85,B 0,C 180,E1 -18841.388,E2 -18841.388} C_VEL
LIN {X 0,Y 272.501,Z 534.936,A -85,B 0,C 180,E1 -18842.572,E2 -18842.572} C_VEL
LIN {X 0,Y 274.702,Z 522.202,A -85,B 0,C 180,E1 -18843.48,E2 -18843.48} C_VEL
LIN {X 0,Y 276.514,Z 507.903,A -85,B 0,C 180,E1 -18844.216,E2 -18844.216} C_VEL
LIN {X 0,Y 277.519,Z 494.136,A -85,B 0,C 180,E1 -18844.68,E2 -18844.68} C_VEL
LIN {X 0,Y 280.787,Z 422.218,A -85,B 0,C 180,E1 -18846.46,E2 -18846.46} C_VEL
LIN {X 0,Y 279.58,Z 414.686,A -85,B 0,C 180,E1 -18846.904,E2 -18846.904} C_VEL
LIN {X 0,Y 271.93,Z 397.711,A -85,B 0,C 180,E1 -18848.819,E2 -18848.819} C_VEL
LIN {X 0,Y 265.487,Z 385.139,A -85,B 0,C 180,E1 -18850.504,E2 -18850.504} C_VEL
LIN {X 0,Y 257.855,Z 371.817,A -85,B 0,C 180,E1 -18852.617,E2 -18852.617} C_VEL
LIN {X 0,Y 254.142,Z 366.048,A -85,B 0,C 180,E1 -18853.693,E2 -18853.693} C_VEL
LIN {X 0,Y 251.704,Z 361.839,A -85,B 0,C 180,E1 -18854.459,E2 -18854.459} C_VEL
LIN {X 0,Y 249.01,Z 353.09,A -85,B 0,C 180,E1 -18858.99,E2 -18858.99} C_VEL
LIN {X 0,Y 249.043,Z 353.089,A -85,B 0,C 180,E1 -18863.657,E2 -18863.657} C_VEL
LIN {X 0,Y 249.024,Z 353.076,A -85,B 0,C 180,E1 -18867.848,E2 -18867.848} C_VEL
LIN {X 0,Y 249.032,Z 353.058,A -85,B 0,C 180,E1 -18871.331,E2 -18871.331} C_VEL
LIN {X 0,Y 249.095,Z 353.072,A -85,B 0,C 180,E1 -18874.963,E2 -18874.963} C_VEL
LIN {X 0,Y 249.082,Z 353.076,A -85,B 0,C 180,E1 -18878.605,E2 -18878.605} C_VEL
LIN {X 0,Y 249.189,Z 353.059,A -85,B 0,C 180,E1 -18883.619,E2 -18883.619} C_VEL
LIN {X 0,Y 249.217,Z 353.053,A -85,B 0,C 180,E1 -18888.615,E2 -18888.615} C_VEL
LIN {X 0,Y 249.406,Z 353.036,A -85,B 0,C 180,E1 -18891.901,E2 -18891.901} C_VEL
LIN {X 0,Y 249.253,Z 353.062,A -85,B 0,C 180,E1 -18895.148,E2 -18895.148} C_VEL
LIN {X 0,Y 249.652,Z 353,A -85,B 0,C 180,E1 -18898.387,E2 -18898.387} C_VEL
LIN {X 0,Y 249.651,Z 353.004,A -85,B 0,C 180,E1 -18901.614,E2 -18901.614} C_VEL
LIN {X 0,Y 249.416,Z 353.032,A -85,B 0,C 180,E1 -18906.678,E2 -18906.678} C_VEL
LIN {X 0,Y 249.328,Z 353.054,A -85,B 0,C 180,E1 -18909.738,E2 -18909.738} C_VEL
LIN {X 0,Y 249.165,Z 353.074,A -85,B 0,C 180,E1 -18914.706,E2 -18914.706} C_VEL
LIN {X 0,Y 249.089,Z 353.082,A -85,B 0,C 180,E1 -18918.082,E2 -18918.082} C_VEL
LIN {X 0,Y 249.07,Z 353.078,A -85,B 0,C 180,E1 -18921.52,E2 -18921.52} C_VEL
LIN {X 0,Y 249.113,Z 353.075,A -85,B 0,C 180,E1 -18925.476,E2 -18925.476} C_VEL
LIN {X 0,Y 249.076,Z 353.079,A -85,B 0,C 180,E1 -18928.993,E2 -18928.993} C_VEL
LIN {X 0,Y 249.027,Z 353.086,A -85,B 0,C 180,E1 -18932.427,E2 -18932.427} C_VEL
LIN {X 0,Y 249.045,Z 353.085,A -85,B 0,C 180,E1 -18936.344,E2 -18936.344} C_VEL
LIN {X 0,Y 249.032,Z 353.159,A -85,B 0,C 180,E1 -18938.963,E2 -18938.963} C_VEL
LIN {X 0,Y 249.961,Z 355.801,A -85,B 0,C 180,E1 -18939.309,E2 -18939.309} C_VEL
LIN {X 0,Y 251.988,Z 358.018,A -85,B 0,C 180,E1 -18939.903,E2 -18939.903} C_VEL
LIN {X 0,Y 254.634,Z 362.02,A -85,B 0,C 180,E1 -18940.698,E2 -18940.698} C_VEL
LIN {X 0,Y 256.124,Z 364.071,A -85,B 0,C 180,E1 -18941.126,E2 -18941.126} C_VEL
LIN {X 0,Y 260.641,Z 370.614,A -85,B 0,C 180,E1 -18942.386,E2 -18942.386} C_VEL
LIN {X 0,Y 268.248,Z 383.434,A -85,B 0,C 180,E1 -18944.419,E2 -18944.419} C_VEL
LIN {X 0,Y 275.966,Z 398.212,A -85,B 0,C 180,E1 -18946.365,E2 -18946.365} C_VEL
LIN {X 0,Y 281.31,Z 409.979,A -85,B 0,C 180,E1 -18947.669,E2 -18947.669} C_VEL
LIN {X 0,Y 277.608,Z 488.253,A -85,B 0,C 180,E1 -18949.63,E2 -18949.63} C_VEL
LIN {X 0,Y 276.255,Z 502.676,A -85,B 0,C 180,E1 -18950.26,E2 -18950.26} C_VEL
LIN {X 0,Y 274.43,Z 516.335,A -85,B 0,C 180,E1 -18951.14,E2 -18951.14} C_VEL
LIN {X 0,Y 272.262,Z 528.636,A -85,B 0,C 180,E1 -18952.19,E2 -18952.19} C_VEL
LIN {X 0,Y 269.353,Z 541.818,A -85,B 0,C 180,E1 -18953.635,E2 -18953.635} C_VEL
LIN {X 0,Y 266.423,Z 553.216,A -85,B 0,C 180,E1 -18955.22,E2 -18955.22} C_VEL
LIN {X 0,Y 263.571,Z 562.91,A -85,B 0,C 180,E1 -18956.865,E2 -18956.865} C_VEL
LIN {X 0,Y 260.274,Z 573.645,A -85,B 0,C 180,E1 -18959.134,E2 -18959.134} C_VEL
LIN {X 0,Y 257.508,Z 582.474,A -85,B 0,C 180,E1 -18961.471,E2 -18961.471} C_VEL
LIN {X 0,Y 254.472,Z 590.903,A -85,B 0,C 180,E1 -18964.217,E2 -18964.217} C_VEL
LIN {X 0,Y 252.097,Z 597.645,A -85,B 0,C 180,E1 -18967.028,E2 -18967.028} C_VEL
LIN {X 0,Y 249.921,Z 603.589,A -85,B 0,C 180,E1 -18970.279,E2 -18970.279} C_VEL
LIN {X 0,Y 248.444,Z 607.924,A -85,B 0,C 180,E1 -18973.568,E2 -18973.568} C_VEL
LIN {X 0,Y 247.434,Z 610.789,A -85,B 0,C 180,E1 -18976.866,E2 -18976.866} C_VEL
LIN {X 0,Y 246.907,Z 612.276,A -85,B 0,C 180,E1 -18980.167,E2 -18980.167} C_VEL
LIN {X 0,Y 246.89,Z 612.427,A -85,B 0,C 180,E1 -18983.462,E2 -18983.462} C_VEL
LIN {X 0,Y 246.925,Z 612.008,A -85,B 0,C 180,E1 -18985.102,E2 -18985.102} C_VEL
LIN {X 0,Y 247.046,Z 610.186,A -85,B 0,C 180,E1 -18988.37,E2 -18988.37} C_VEL
LIN {X 0,Y 247.346,Z 607.009,A -85,B 0,C 180,E1 -18991.628,E2 -18991.628} C_VEL
LIN {X 0,Y 248.11,Z 602.35,A -85,B 0,C 180,E1 -18994.875,E2 -18994.875} C_VEL
LIN {X 0,Y 249.459,Z 596.074,A -85,B 0,C 180,E1 -18998.098,E2 -18998.098} C_VEL
LIN {X 0,Y 251.235,Z 589.083,A -85,B 0,C 180,E1 -19000.884,E2 -19000.884} C_VEL
LIN {X 0,Y 253.294,Z 580.816,A -85,B 0,C 180,E1 -19003.526,E2 -19003.526} C_VEL
LIN {X 0,Y 255.395,Z 571.419,A -85,B 0,C 180,E1 -19005.972,E2 -19005.972} C_VEL
LIN {X 0,Y 257.931,Z 560.479,A -85,B 0,C 180,E1 -19008.26,E2 -19008.26} C_VEL
LIN {X 0,Y 260.323,Z 549.324,A -85,B 0,C 180,E1 -19010.133,E2 -19010.133} C_VEL
LIN {X 0,Y 262.628,Z 537.002,A -85,B 0,C 180,E1 -19011.795,E2 -19011.795} C_VEL
LIN {X 0,Y 264.587,Z 525.141,A -85,B 0,C 180,E1 -19013.065,E2 -19013.065} C_VEL
LIN {X 0,Y 266.297,Z 512.183,A -85,B 0,C 180,E1 -19014.146,E2 -19014.146} C_VEL
LIN {X 0,Y 267.753,Z 498.215,A -85,B 0,C 180,E1 -19014.987,E2 -19014.987} C_VEL
LIN {X 0,Y 268.609,Z 485.076,A -85,B 0,C 180,E1 -19015.524,E2 -19015.524} C_VEL
LIN {X 0,Y 271.626,Z 400.501,A -85,B 0,C 180,E1 -19017.727,E2 -19017.727} C_VEL
LIN {X 0,Y 265.092,Z 384.313,A -85,B 0,C 180,E1 -19019.1,E2 -19019.1} C_VEL
LIN {X 0,Y 258.322,Z 369.76,A -85,B 0,C 180,E1 -19020.546,E2 -19020.546} C_VEL
LIN {X 0,Y 252.738,Z 360.18,A -85,B 0,C 180,E1 -19021.734,E2 -19021.734} C_VEL
LIN {X 0,Y 250.643,Z 356.778,A -85,B 0,C 180,E1 -19022.191,E2 -19022.191} C_VEL
LIN {X 0,Y 249.277,Z 354.259,A -85,B 0,C 180,E1 -19022.505,E2 -19022.505} C_VEL
LIN {X 0,Y 249.024,Z 353.089,A -85,B 0,C 180,E1 -19022.605,E2 -19022.605} C_VEL
LIN {X 0,Y 249.07,Z 353.074,A -85,B 0,C 180,E1 -19026.337,E2 -19026.337} C_VEL
LIN {X 0,Y 249.025,Z 353.068,A -85,B 0,C 180,E1 -19030.473,E2 -19030.473} C_VEL
LIN {X 0,Y 248.992,Z 353.088,A -85,B 0,C 180,E1 -19034.88,E2 -19034.88} C_VEL
LIN {X 0,Y 249.008,Z 353.089,A -85,B 0,C 180,E1 -19037.36,E2 -19037.36} C_VEL
LIN {X 0,Y 249.023,Z 353.083,A -85,B 0,C 180,E1 -19041.618,E2 -19041.618} C_VEL
LIN {X 0,Y 249.04,Z 353.083,A -85,B 0,C 180,E1 -19045.638,E2 -19045.638} C_VEL
LIN {X 0,Y 249.041,Z 353.088,A -85,B 0,C 180,E1 -19049.471,E2 -19049.471} C_VEL
LIN {X 0,Y 249.055,Z 353.067,A -85,B 0,C 180,E1 -19053.159,E2 -19053.159} C_VEL
LIN {X 0,Y 249.05,Z 353.086,A -85,B 0,C 180,E1 -19056.729,E2 -19056.729} C_VEL
LIN {X 0,Y 249.052,Z 353.063,A -85,B 0,C 180,E1 -19060.206,E2 -19060.206} C_VEL
LIN {X 0,Y 249.152,Z 353.073,A -85,B 0,C 180,E1 -19063.615,E2 -19063.615} C_VEL
LIN {X 0,Y 249.223,Z 353.045,A -85,B 0,C 180,E1 -19068.615,E2 -19068.615} C_VEL
LIN {X 0,Y 249.409,Z 353.036,A -85,B 0,C 180,E1 -19072.356,E2 -19072.356} C_VEL
LIN {X 0,Y 248.738,Z 353.112,A -85,B 0,C 180,E1 -19073.703,E2 -19073.703} C_VEL
LIN {X 0,Y 245.957,Z 353.453,A -85,B 0,C 180,E1 -19075.902,E2 -19075.902} C_VEL
LIN {X 0,Y 243.629,Z 353.753,A -85,B 0,C 180,E1 -19077.693,E2 -19077.693} C_VEL
LIN {X 0,Y 242.663,Z 353.883,A -85,B 0,C 180,E1 -19079.079,E2 -19079.079} C_VEL
LIN {X 0,Y 242.6,Z 353.887,A -85,B 0,C 180,E1 -19079.548,E2 -19079.548} C_VEL
LIN {X 0,Y 242.6,Z 353.881,A -85,B 0,C 180,E1 -19081.66,E2 -19081.66} C_VEL
LIN {X 0,Y 242.386,Z 353.917,A -85,B 0,C 180,E1 -19086.66,E2 -19086.66} C_VEL
LIN {X 0,Y 242.254,Z 353.917,A -85,B 0,C 180,E1 -19090.024,E2 -19090.024} C_VEL
LIN {X 0,Y 242.129,Z 353.935,A -85,B 0,C 180,E1 -19095.143,E2 -19095.143} C_VEL
LIN {X 0,Y 242.042,Z 353.959,A -85,B 0,C 180,E1 -19098.626,E2 -19098.626} C_VEL
LIN {X 0,Y 241.996,Z 353.953,A -85,B 0,C 180,E1 -19102.181,E2 -19102.181} C_VEL
LIN {X 0,Y 242.026,Z 353.95,A -85,B 0,C 180,E1 -19105.821,E2 -19105.821} C_VEL
LIN {X 0,Y 241.962,Z 353.964,A -85,B 0,C 180,E1 -19109.589,E2 -19109.589} C_VEL
LIN {X 0,Y 241.974,Z 353.965,A -85,B 0,C 180,E1 -19113.493,E2 -19113.493} C_VEL
LIN {X 0,Y 241.987,Z 353.962,A -85,B 0,C 180,E1 -19117.582,E2 -19117.582} C_VEL
LIN {X 0,Y 241.932,Z 353.956,A -85,B 0,C 180,E1 -19121.923,E2 -19121.923} C_VEL
LIN {X 0,Y 241.93,Z 353.973,A -85,B 0,C 180,E1 -19126.572,E2 -19126.572} C_VEL
LIN {X 0,Y 241.972,Z 354.088,A -85,B 0,C 180,E1 -19126.998,E2 -19126.998} C_VEL
LIN {X 0,Y 244.261,Z 362.383,A -85,B 0,C 180,E1 -19130.548,E2 -19130.548} C_VEL
LIN {X 0,Y 251.852,Z 377.679,A -85,B 0,C 180,E1 -19132.359,E2 -19132.359} C_VEL
LIN {X 0,Y 258.725,Z 393.046,A -85,B 0,C 180,E1 -19133.913,E2 -19133.913} C_VEL
LIN {X 0,Y 263.025,Z 404.173,A -85,B 0,C 180,E1 -19134.879,E2 -19134.879} C_VEL
LIN {X 0,Y 265.055,Z 419.435,A -85,B 0,C 180,E1 -19135.634,E2 -19135.634} C_VEL
LIN {X 0,Y 261.816,Z 501.384,A -85,B 0,C 180,E1 -19137.815,E2 -19137.815} C_VEL
LIN {X 0,Y 260.598,Z 515.172,A -85,B 0,C 180,E1 -19138.443,E2 -19138.443} C_VEL
LIN {X 0,Y 258.8,Z 529.318,A -85,B 0,C 180,E1 -19139.392,E2 -19139.392} C_VEL
LIN {X 0,Y 256.863,Z 541.54,A -85,B 0,C 180,E1 -19140.496,E2 -19140.496} C_VEL
LIN {X 0,Y 254.52,Z 554.414,A -85,B 0,C 180,E1 -19142.004,E2 -19142.004} C_VEL
LIN {X 0,Y 251.966,Z 566.102,A -85,B 0,C 180,E1 -19143.718,E2 -19143.718} C_VEL
LIN {X 0,Y 249.731,Z 575.83,A -85,B 0,C 180,E1 -19145.475,E2 -19145.475} C_VEL
LIN {X 0,Y 247.138,Z 586.614,A -85,B 0,C 180,E1 -19147.865,E2 -19147.865} C_VEL
LIN {X 0,Y 244.971,Z 595.511,A -85,B 0,C 180,E1 -19150.301,E2 -19150.301} C_VEL
LIN {X 0,Y 243.102,Z 604.042,A -85,B 0,C 180,E1 -19153.197,E2 -19153.197} C_VEL
LIN {X 0,Y 241.772,Z 609.979,A -85,B 0,C 180,E1 -19155.695,E2 -19155.695} C_VEL
LIN {X 0,Y 240.532,Z 616.315,A -85,B 0,C 180,E1 -19159.052,E2 -19159.052} C_VEL
LIN {X 0,Y 240.118,Z 619.929,A -85,B 0,C 180,E1 -19161.585,E2 -19161.585} C_VEL
LIN {X 0,Y 239.835,Z 623.566,A -85,B 0,C 180,E1 -19165.079,E2 -19165.079} C_VEL
LIN {X 0,Y 239.841,Z 625.572,A -85,B 0,C 180,E1 -19168.321,E2 -19168.321} C_VEL
LIN {X 0,Y 239.913,Z 626.116,A -85,B 0,C 180,E1 -19170,E2 -19170} C_VEL
LIN {X 0,Y 239.754,Z 626.186,A -85,B 0,C 180,E1 -19173.361,E2 -19173.361} C_VEL
LIN {X 0,Y 239.892,Z 624.929,A -85,B 0,C 180,E1 -19176.73,E2 -19176.73} C_VEL
LIN {X 0,Y 240.471,Z 622.32,A -85,B 0,C 180,E1 -19180.099,E2 -19180.099} C_VEL
LIN {X 0,Y 241.567,Z 618.28,A -85,B 0,C 180,E1 -19183.458,E2 -19183.458} C_VEL
LIN {X 0,Y 242.983,Z 614.262,A -85,B 0,C 180,E1 -19185.948,E2 -19185.948} C_VEL
LIN {X 0,Y 245.186,Z 607.648,A -85,B 0,C 180,E1 -19189.159,E2 -19189.159} C_VEL
LIN {X 0,Y 248.009,Z 599.89,A -85,B 0,C 180,E1 -19192.053,E2 -19192.053} C_VEL
LIN {X 0,Y 250.815,Z 592.038,A -85,B 0,C 180,E1 -19194.412,E2 -19194.412} C_VEL
LIN {X 0,Y 254.092,Z 582.585,A -85,B 0,C 180,E1 -19196.708,E2 -19196.708} C_VEL
LIN {X 0,Y 257.76,Z 571.073,A -85,B 0,C 180,E1 -19198.944,E2 -19198.944} C_VEL
LIN {X 0,Y 260.713,Z 560.498,A -85,B 0,C 180,E1 -19200.607,E2 -19200.607} C_VEL
LIN {X 0,Y 263.854,Z 547.889,A -85,B 0,C 180,E1 -19202.188,E2 -19202.188} C_VEL
LIN {X 0,Y 266.575,Z 535.458,A -85,B 0,C 180,E1 -19203.39,E2 -19203.39} C_VEL
LIN {X 0,Y 268.848,Z 522.947,A -85,B 0,C 180,E1 -19204.309,E2 -19204.309} C_VEL
LIN {X 0,Y 270.678,Z 509.042,A -85,B 0,C 180,E1 -19205.061,E2 -19205.061} C_VEL
LIN {X 0,Y 271.759,Z 496.124,A -85,B 0,C 180,E1 -19205.525,E2 -19205.525} C_VEL
LIN {X 0,Y 275.202,Z 423.898,A -85,B 0,C 180,E1 -19207.347,E2 -19207.347} C_VEL
LIN {X 0,Y 274.305,Z 417.553,A -85,B 0,C 180,E1 -19207.716,E2 -19207.716} C_VEL
